SPLINE
SPL {X  -156.487, Y  +349.204, Z    +0.000, E1   +21.338, E3 +359209.083}
SPL {X  -159.136, Y  +365.992, Z    +0.000, E1   +12.463, E3 +359219.841}
SPL {X  -159.799, Y  +374.694, Z    +0.000, E1    +7.504, E3 +359222.945}
SPL {X  -159.976, Y  +380.404, Z    +0.000, E1    +3.959, E3 +359224.478}
SPL {X  -159.990, Y  +384.773, Z    +0.000, E1    +1.003, E3 +359225.373}
SPL {X  -159.990, Y  +387.968, Z    +0.000, E1    -1.448, E3 +359225.941}
SPL {X  -159.990, Y  +391.397, Z    +0.000, E1    -4.422, E3 +359226.565}
SPL {X  -159.990, Y  +395.864, Z    +0.000, E1    -8.712, E3 +359227.653}
SPL {X  -159.990, Y  +401.273, Z    +0.000, E1   -14.176, E3 +359229.381}
SPL {X  -159.990, Y  +411.788, Z    +0.000, E1   -23.693, E3 +359234.924}
SPL {X  -159.990, Y  +438.158, Z    +0.000, E1   -37.630, E3 +359258.201}
SPL {X  -159.990, Y  +468.567, Z    +0.000, E1   -41.922, E3 +359307.545}
SPL {X  -159.990, Y  +474.616, Z    +0.000, E1   -41.909, E3 +359321.874}
SPL {X  -159.990, Y  +478.952, Z    +0.000, E1   -41.885, E3 +359332.172}
SPL {X  -159.990, Y  +484.724, Z    +0.000, E1   -41.943, E3 +359345.724}
SPL {X  -159.990, Y  +492.944, Z    +0.000, E1   -41.952, E3 +359365.143}
SPL {X  -159.990, Y  +499.538, Z    +0.000, E1   -41.904, E3 +359380.802}
SPL {X  -159.990, Y  +504.097, Z    +0.000, E1   -41.897, E3 +359391.590}
SPL {X  -159.990, Y  +509.413, Z    +0.000, E1   -41.921, E3 +359404.126}
SPL {X  -159.990, Y  +516.193, Z    +0.000, E1   -41.932, E3 +359420.142}
SPL {X  -159.990, Y  +521.318, Z    +0.000, E1   -41.891, E3 +359432.316}
SPL {X  -159.990, Y  +526.974, Z    +0.000, E1   -41.950, E3 +359445.605}
SPL {X  -159.990, Y  +533.758, Z    +0.000, E1   -41.910, E3 +359461.708}
SPL {X  -159.990, Y  +539.474, Z    +0.000, E1   -41.912, E3 +359475.235}
SPL {X  -159.990, Y  +544.879, Z    +0.000, E1   -41.899, E3 +359488.046}
SPL {X  -159.990, Y  +550.802, Z    +0.000, E1   -41.920, E3 +359502.028}
SPL {X  -159.990, Y  +556.952, Z    +0.000, E1   -41.911, E3 +359516.567}
SPL {X  -159.990, Y  +562.629, Z    +0.000, E1   -41.910, E3 +359529.985}
SPL {X  -159.990, Y  +567.682, Z    +0.000, E1   -41.901, E3 +359541.944}
SPL {X  -159.990, Y  +572.912, Z    +0.000, E1   -41.914, E3 +359554.291}
SPL {X  -159.990, Y  +578.863, Z    +0.000, E1   -41.918, E3 +359568.355}
SPL {X  -159.990, Y  +584.320, Z    +0.000, E1   -41.901, E3 +359581.302}
SPL {X  -159.990, Y  +589.217, Z    +0.000, E1   -41.901, E3 +359592.875}
SPL {X  -159.990, Y  +594.252, Z    +0.000, E1   -41.903, E3 +359604.789}
SPL {X  -159.990, Y  +600.237, Z    +0.000, E1   -41.928, E3 +359618.907}
SPL {X  -159.990, Y  +605.518, Z    +0.000, E1   -41.890, E3 +359631.445}
SPL {X  -159.990, Y  +610.545, Z    +0.000, E1   -41.917, E3 +359643.293}
SPL {X  -159.990, Y  +615.720, Z    +0.000, E1   -41.899, E3 +359655.553}
SPL {X  -159.990, Y  +621.417, Z    +0.000, E1   -41.931, E3 +359668.990}
SPL {X  -159.990, Y  +627.900, Z    +0.000, E1   -41.914, E3 +359684.330}
SPL {X  -159.990, Y  +632.270, Z    +0.000, E1   -41.887, E3 +359694.706}
SPL {X  -159.990, Y  +637.009, Z    +0.000, E1   -41.925, E3 +359705.848}
SPL {X  -159.990, Y  +642.624, Z    +0.000, E1   -41.901, E3 +359719.169}
SPL {X  -159.990, Y  +647.782, Z    +0.000, E1   -41.914, E3 +359731.337}
SPL {X  -159.990, Y  +653.094, Z    +0.000, E1   -41.905, E3 +359743.916}
SPL {X  -159.990, Y  +657.893, Z    +0.000, E1   -41.899, E3 +359755.281}
SPL {X  -159.990, Y  +662.516, Z    +0.000, E1   -41.899, E3 +359766.213}
SPL {X  -159.990, Y  +666.974, Z    +0.000, E1   -41.897, E3 +359776.757}
SPL {X  -159.984, Y  +672.859, Z    +0.000, E1   -41.934, E3 +359790.618}
SPL {X  -159.817, Y  +678.937, Z    +0.000, E1   -41.879, E3 +359805.206}
SPL {X  -159.484, Y  +684.213, Z    +0.000, E1   -41.818, E3 +359818.043}
SPL {X  -159.007, Y  +689.209, Z    +0.000, E1   -41.732, E3 +359830.347}
SPL {X  -158.327, Y  +694.511, Z    +0.000, E1   -41.622, E3 +359843.598}
SPL {X  -157.480, Y  +699.729, Z    +0.000, E1   -41.453, E3 +359856.861}
SPL {X  -156.604, Y  +704.242, Z    +0.000, E1   -41.288, E3 +359868.470}
SPL {X  -155.514, Y  +709.078, Z    +0.000, E1   -41.107, E3 +359881.024}
SPL {X  -154.232, Y  +714.035, Z    +0.000, E1   -40.861, E3 +359894.083}
SPL {X  -153.147, Y  +717.790, Z    +0.000, E1   -40.640, E3 +359904.101}
SPL {X  -151.881, Y  +721.788, Z    +0.000, E1   -40.435, E3 +359914.787}
SPL {X  -148.572, Y  +730.857, Z    +0.000, E1   -36.304, E3 +359970.996}
ENDSPLINE

SPLINE
SPL {X  -156.377, Y  +705.307, Z    +0.000, E1   -21.740, E3 +360025.245}
SPL {X  -158.965, Y  +689.585, Z    +0.000, E1   -13.405, E3 +360036.403}
SPL {X  -159.884, Y  +677.314, Z    +0.000, E1    -6.475, E3 +360041.115}
SPL {X  -159.990, Y  +670.142, Z    +0.000, E1    -1.740, E3 +360042.905}
SPL {X  -159.990, Y  +666.629, Z    +0.000, E1    +0.827, E3 +360043.554}
SPL {X  -159.990, Y  +662.407, Z    +0.000, E1    +4.406, E3 +360044.405}
SPL {X  -159.990, Y  +655.884, Z    +0.000, E1   +10.601, E3 +360046.270}
SPL {X  -159.990, Y  +643.833, Z    +0.000, E1   +21.883, E3 +360051.899}
SPL {X  -159.990, Y  +617.235, Z    +0.000, E1   +36.481, E3 +360075.799}
SPL {X  -159.990, Y  +586.905, Z    +0.000, E1   +41.264, E3 +360124.776}
SPL {X  -159.990, Y  +581.111, Z    +0.000, E1   +41.245, E3 +360138.829}
SPL {X  -159.990, Y  +576.269, Z    +0.000, E1   +41.239, E3 +360150.557}
SPL {X  -159.990, Y  +571.714, Z    +0.000, E1   +41.240, E3 +360161.585}
SPL {X  -159.990, Y  +567.050, Z    +0.000, E1   +41.238, E3 +360172.872}
SPL {X  -159.990, Y  +561.959, Z    +0.000, E1   +41.251, E3 +360185.170}
SPL {X  -159.990, Y  +557.719, Z    +0.000, E1   +41.226, E3 +360195.473}
SPL {X  -159.990, Y  +554.148, Z    +0.000, E1   +41.237, E3 +360204.088}
SPL {X  -159.990, Y  +548.812, Z    +0.000, E1   +41.263, E3 +360216.963}
SPL {X  -159.990, Y  +543.804, Z    +0.000, E1   +41.237, E3 +360229.127}
SPL {X  -159.990, Y  +538.952, Z    +0.000, E1   +41.247, E3 +360240.875}
SPL {X  -159.990, Y  +534.225, Z    +0.000, E1   +41.236, E3 +360252.308}
SPL {X  -159.990, Y  +529.136, Z    +0.000, E1   +41.262, E3 +360264.584}
SPL {X  -159.990, Y  +522.690, Z    +0.000, E1   +41.265, E3 +360280.183}
SPL {X  -159.990, Y  +516.698, Z    +0.000, E1   +41.259, E3 +360294.658}
SPL {X  -159.990, Y  +510.896, Z    +0.000, E1   +41.267, E3 +360308.675}
SPL {X  -159.990, Y  +505.215, Z    +0.000, E1   +41.261, E3 +360322.435}
SPL {X  -159.990, Y  +500.102, Z    +0.000, E1   +41.251, E3 +360334.819}
SPL {X  -159.990, Y  +495.023, Z    +0.000, E1   +41.263, E3 +360347.067}
SPL {X  -159.990, Y  +479.011, Z    +0.000, E1   +45.740, E3 +360356.449}
SPL {X  -159.990, Y  +471.379, Z    +0.000, E1   +46.435, E3 +360368.065}
SPL {X  -159.990, Y  +466.895, Z    +0.000, E1   +45.533, E3 +360382.470}
SPL {X  -159.990, Y  +462.409, Z    +0.000, E1   +44.664, E3 +360397.245}
SPL {X  -159.990, Y  +458.229, Z    +0.000, E1   +43.579, E3 +360412.727}
SPL {X  -159.990, Y  +453.434, Z    +0.000, E1   +43.227, E3 +360425.501}
SPL {X  -159.990, Y  +448.702, Z    +0.000, E1   +43.218, E3 +360436.223}
SPL {X  -159.990, Y  +444.476, Z    +0.000, E1   +43.219, E3 +360445.761}
SPL {X  -159.990, Y  +440.246, Z    +0.000, E1   +43.217, E3 +360455.319}
SPL {X  -159.990, Y  +434.411, Z    +0.000, E1   +43.246, E3 +360468.449}
SPL {X  -159.990, Y  +429.216, Z    +0.000, E1   +43.210, E3 +360480.222}
SPL {X  -159.990, Y  +424.433, Z    +0.000, E1   +43.237, E3 +360490.970}
SPL {X  -159.990, Y  +419.466, Z    +0.000, E1   +43.217, E3 +360502.209}
SPL {X  -159.990, Y  +414.585, Z    +0.000, E1   +43.233, E3 +360513.201}
SPL {X  -159.990, Y  +409.927, Z    +0.000, E1   +43.217, E3 +360523.733}
SPL {X  -159.990, Y  +405.428, Z    +0.000, E1   +43.230, E3 +360533.891}
SPL {X  -159.990, Y  +398.518, Z    +0.000, E1   +43.261, E3 +360549.445}
SPL {X  -159.990, Y  +392.163, Z    +0.000, E1   +43.223, E3 +360563.845}
SPL {X  -159.990, Y  +387.342, Z    +0.000, E1   +43.224, E3 +360574.723}
SPL {X  -159.990, Y  +382.548, Z    +0.000, E1   +43.224, E3 +360585.546}
SPL {X  -159.922, Y  +377.835, Z    +0.000, E1   +43.211, E3 +360596.262}
SPL {X  -159.712, Y  +373.072, Z    +0.000, E1   +43.177, E3 +360607.228}
SPL {X  -159.289, Y  +367.537, Z    +0.000, E1   +43.118, E3 +360620.140}
SPL {X  -158.730, Y  +362.464, Z    +0.000, E1   +43.003, E3 +360632.172}
SPL {X  -158.182, Y  +358.518, Z    +0.000, E1   +42.902, E3 +360641.650}
SPL {X  -157.507, Y  +354.423, Z    +0.000, E1   +42.786, E3 +360651.596}
SPL {X  -156.676, Y  +350.104, Z    +0.000, E1   +42.637, E3 +360662.201}
SPL {X  -155.807, Y  +346.154, Z    +0.000, E1   +42.470, E3 +360672.028}
SPL {X  -154.777, Y  +341.993, Z    +0.000, E1   +42.302, E3 +360682.453}
SPL {X  -153.585, Y  +337.686, Z    +0.000, E1   +42.062, E3 +360693.429}
SPL {X  -152.412, Y  +333.846, Z    +0.000, E1   +41.856, E3 +360703.271}
SPL {X  -151.009, Y  +329.651, Z    +0.000, E1   +41.581, E3 +360714.171}
SPL {X  -148.356, Y  +322.607, Z    +0.000, E1   +36.121, E3 +360774.647}
ENDSPLINE

SPLINE
SPL {X  -156.487, Y  +349.204, Z    +0.000, E1   +21.338, E3 +360829.773}
SPL {X  -159.136, Y  +365.992, Z    +0.000, E1   +12.463, E3 +360840.531}
SPL {X  -159.799, Y  +374.694, Z    +0.000, E1    +7.504, E3 +360843.635}
SPL {X  -159.976, Y  +380.404, Z    +0.000, E1    +3.959, E3 +360845.168}
SPL {X  -159.990, Y  +384.773, Z    +0.000, E1    +1.003, E3 +360846.062}
SPL {X  -159.990, Y  +387.968, Z    +0.000, E1    -1.448, E3 +360846.631}
SPL {X  -159.990, Y  +391.397, Z    +0.000, E1    -4.422, E3 +360847.255}
SPL {X  -159.990, Y  +395.864, Z    +0.000, E1    -8.712, E3 +360848.343}
SPL {X  -159.990, Y  +401.273, Z    +0.000, E1   -14.176, E3 +360850.070}
SPL {X  -159.990, Y  +409.369, Z    +0.000, E1   -21.807, E3 +360853.862}
SPL {X  -159.990, Y  +436.107, Z    +0.000, E1   -36.921, E3 +360876.787}
SPL {X  -159.990, Y  +465.724, Z    +0.000, E1   -41.883, E3 +360921.586}
SPL {X  -159.990, Y  +470.837, Z    +0.000, E1   -41.927, E3 +360933.600}
SPL {X  -159.990, Y  +477.498, Z    +0.000, E1   -41.916, E3 +360949.375}
SPL {X  -159.990, Y  +483.140, Z    +0.000, E1   -41.902, E3 +360962.731}
SPL {X  -159.990, Y  +488.618, Z    +0.000, E1   -41.913, E3 +360975.663}
SPL {X  -159.990, Y  +494.299, Z    +0.000, E1   -41.910, E3 +360989.097}
SPL {X  -159.990, Y  +499.538, Z    +0.000, E1   -41.904, E3 +361001.491}
SPL {X  -159.990, Y  +505.259, Z    +0.000, E1   -41.922, E3 +361014.991}
SPL {X  -159.990, Y  +511.862, Z    +0.000, E1   -41.927, E3 +361030.601}
SPL {X  -159.990, Y  +519.146, Z    +0.000, E1   -41.942, E3 +361047.795}
SPL {X  -159.990, Y  +526.974, Z    +0.000, E1   -41.950, E3 +361066.295}
SPL {X  -159.990, Y  +533.758, Z    +0.000, E1   -41.910, E3 +361082.397}
SPL {X  -159.990, Y  +539.474, Z    +0.000, E1   -41.912, E3 +361095.925}
SPL {X  -159.990, Y  +544.879, Z    +0.000, E1   -41.899, E3 +361108.736}
SPL {X  -159.990, Y  +550.802, Z    +0.000, E1   -41.920, E3 +361122.717}
SPL {X  -159.990, Y  +556.952, Z    +0.000, E1   -41.911, E3 +361137.257}
SPL {X  -159.990, Y  +562.629, Z    +0.000, E1   -41.910, E3 +361150.675}
SPL {X  -159.990, Y  +567.682, Z    +0.000, E1   -41.901, E3 +361162.634}
SPL {X  -159.990, Y  +572.912, Z    +0.000, E1   -41.914, E3 +361174.981}
SPL {X  -159.990, Y  +578.863, Z    +0.000, E1   -41.918, E3 +361189.045}
SPL {X  -159.990, Y  +584.320, Z    +0.000, E1   -41.901, E3 +361201.992}
SPL {X  -159.990, Y  +589.217, Z    +0.000, E1   -41.901, E3 +361213.564}
SPL {X  -159.990, Y  +594.252, Z    +0.000, E1   -41.903, E3 +361225.479}
SPL {X  -159.990, Y  +598.793, Z    +0.000, E1   -41.896, E3 +361236.233}
SPL {X  -159.990, Y  +604.215, Z    +0.000, E1   -41.919, E3 +361249.013}
SPL {X  -159.990, Y  +609.216, Z    +0.000, E1   -41.890, E3 +361260.881}
SPL {X  -159.990, Y  +614.570, Z    +0.000, E1   -41.926, E3 +361273.486}
SPL {X  -159.990, Y  +620.005, Z    +0.000, E1   -41.900, E3 +361286.376}
SPL {X  -159.990, Y  +624.919, Z    +0.000, E1   -41.912, E3 +361297.983}
SPL {X  -159.990, Y  +630.816, Z    +0.000, E1   -41.915, E3 +361311.912}
SPL {X  -159.990, Y  +637.009, Z    +0.000, E1   -41.925, E3 +361326.538}
SPL {X  -159.990, Y  +642.624, Z    +0.000, E1   -41.901, E3 +361339.858}
SPL {X  -159.990, Y  +647.782, Z    +0.000, E1   -41.914, E3 +361352.027}
SPL {X  -159.990, Y  +653.094, Z    +0.000, E1   -41.905, E3 +361364.605}
SPL {X  -159.990, Y  +657.893, Z    +0.000, E1   -41.899, E3 +361375.971}
SPL {X  -159.990, Y  +662.516, Z    +0.000, E1   -41.899, E3 +361386.902}
SPL {X  -159.990, Y  +666.974, Z    +0.000, E1   -41.897, E3 +361397.447}
SPL {X  -159.984, Y  +672.859, Z    +0.000, E1   -41.934, E3 +361411.308}
SPL {X  -159.817, Y  +678.937, Z    +0.000, E1   -41.879, E3 +361425.896}
SPL {X  -159.484, Y  +684.213, Z    +0.000, E1   -41.818, E3 +361438.732}
SPL {X  -159.007, Y  +689.209, Z    +0.000, E1   -41.732, E3 +361451.037}
SPL {X  -158.327, Y  +694.511, Z    +0.000, E1   -41.622, E3 +361464.288}
SPL {X  -157.480, Y  +699.729, Z    +0.000, E1   -41.453, E3 +361477.551}
SPL {X  -156.604, Y  +704.242, Z    +0.000, E1   -41.288, E3 +361489.160}
SPL {X  -155.514, Y  +709.078, Z    +0.000, E1   -41.107, E3 +361501.713}
SPL {X  -154.232, Y  +714.035, Z    +0.000, E1   -40.861, E3 +361514.772}
SPL {X  -153.147, Y  +717.790, Z    +0.000, E1   -40.640, E3 +361524.791}
SPL {X  -151.881, Y  +721.788, Z    +0.000, E1   -40.435, E3 +361535.477}
SPL {X  -148.572, Y  +730.857, Z    +0.000, E1   -36.304, E3 +361591.686}
ENDSPLINE

SPLINE
SPL {X  -156.377, Y  +705.307, Z    +0.000, E1   -21.740, E3 +361645.935}
SPL {X  -158.965, Y  +689.585, Z    +0.000, E1   -13.405, E3 +361657.092}
SPL {X  -159.884, Y  +677.314, Z    +0.000, E1    -6.475, E3 +361661.805}
SPL {X  -159.990, Y  +670.142, Z    +0.000, E1    -1.740, E3 +361663.594}
SPL {X  -159.990, Y  +666.629, Z    +0.000, E1    +0.827, E3 +361664.244}
SPL {X  -159.990, Y  +662.407, Z    +0.000, E1    +4.406, E3 +361665.094}
SPL {X  -159.990, Y  +655.884, Z    +0.000, E1   +10.601, E3 +361666.960}
SPL {X  -159.990, Y  +643.833, Z    +0.000, E1   +21.883, E3 +361672.589}
SPL {X  -159.990, Y  +617.235, Z    +0.000, E1   +36.481, E3 +361696.489}
SPL {X  -159.990, Y  +586.905, Z    +0.000, E1   +41.264, E3 +361745.465}
SPL {X  -159.990, Y  +581.111, Z    +0.000, E1   +41.245, E3 +361759.519}
SPL {X  -159.990, Y  +576.269, Z    +0.000, E1   +41.239, E3 +361771.247}
SPL {X  -159.990, Y  +571.714, Z    +0.000, E1   +41.240, E3 +361782.275}
SPL {X  -159.990, Y  +567.050, Z    +0.000, E1   +41.238, E3 +361793.561}
SPL {X  -159.990, Y  +561.959, Z    +0.000, E1   +41.251, E3 +361805.860}
SPL {X  -159.990, Y  +555.553, Z    +0.000, E1   +41.273, E3 +361821.328}
SPL {X  -159.990, Y  +549.897, Z    +0.000, E1   +41.240, E3 +361835.058}
SPL {X  -159.990, Y  +544.775, Z    +0.000, E1   +41.260, E3 +361847.433}
SPL {X  -159.990, Y  +538.952, Z    +0.000, E1   +41.247, E3 +361861.564}
SPL {X  -159.990, Y  +534.225, Z    +0.000, E1   +41.236, E3 +361872.997}
SPL {X  -159.990, Y  +529.136, Z    +0.000, E1   +41.262, E3 +361885.273}
SPL {X  -159.990, Y  +524.776, Z    +0.000, E1   +41.225, E3 +361895.887}
SPL {X  -159.990, Y  +521.454, Z    +0.000, E1   +41.236, E3 +361903.909}
SPL {X  -159.990, Y  +515.605, Z    +0.000, E1   +41.288, E3 +361917.948}
SPL {X  -159.990, Y  +509.898, Z    +0.000, E1   +41.246, E3 +361931.809}
SPL {X  -159.990, Y  +505.215, Z    +0.000, E1   +41.261, E3 +361943.125}
SPL {X  -159.990, Y  +500.102, Z    +0.000, E1   +41.251, E3 +361955.508}
SPL {X  -159.990, Y  +495.023, Z    +0.000, E1   +41.263, E3 +361967.757}
SPL {X  -159.990, Y  +479.011, Z    +0.000, E1   +45.740, E3 +361977.139}
SPL {X  -159.990, Y  +471.379, Z    +0.000, E1   +46.435, E3 +361988.754}
SPL {X  -159.990, Y  +465.881, Z    +0.000, E1   +45.385, E3 +362006.357}
SPL {X  -159.990, Y  +461.571, Z    +0.000, E1   +44.440, E3 +362020.883}
SPL {X  -159.990, Y  +458.229, Z    +0.000, E1   +43.579, E3 +362033.416}
SPL {X  -159.990, Y  +453.434, Z    +0.000, E1   +43.227, E3 +362046.191}
SPL {X  -159.990, Y  +448.702, Z    +0.000, E1   +43.218, E3 +362056.913}
SPL {X  -159.990, Y  +442.224, Z    +0.000, E1   +43.270, E3 +362071.463}
SPL {X  -159.990, Y  +435.724, Z    +0.000, E1   +43.218, E3 +362086.221}
SPL {X  -159.990, Y  +430.527, Z    +0.000, E1   +43.236, E3 +362097.910}
SPL {X  -159.990, Y  +424.433, Z    +0.000, E1   +43.237, E3 +362111.659}
SPL {X  -159.990, Y  +419.466, Z    +0.000, E1   +43.217, E3 +362122.899}
SPL {X  -159.990, Y  +414.585, Z    +0.000, E1   +43.233, E3 +362133.891}
SPL {X  -159.990, Y  +409.927, Z    +0.000, E1   +43.217, E3 +362144.422}
SPL {X  -159.990, Y  +405.428, Z    +0.000, E1   +43.230, E3 +362154.581}
SPL {X  -159.990, Y  +401.033, Z    +0.000, E1   +43.209, E3 +362164.535}
SPL {X  -159.990, Y  +396.968, Z    +0.000, E1   +43.221, E3 +362173.693}
SPL {X  -159.990, Y  +392.163, Z    +0.000, E1   +43.223, E3 +362184.535}
SPL {X  -159.990, Y  +387.342, Z    +0.000, E1   +43.224, E3 +362195.412}
SPL {X  -159.990, Y  +382.548, Z    +0.000, E1   +43.224, E3 +362206.235}
SPL {X  -159.922, Y  +377.835, Z    +0.000, E1   +43.211, E3 +362216.952}
SPL {X  -159.712, Y  +373.072, Z    +0.000, E1   +43.177, E3 +362227.918}
SPL {X  -159.289, Y  +367.537, Z    +0.000, E1   +43.118, E3 +362240.830}
SPL {X  -158.730, Y  +362.464, Z    +0.000, E1   +43.003, E3 +362252.862}
SPL {X  -158.182, Y  +358.518, Z    +0.000, E1   +42.902, E3 +362262.340}
SPL {X  -157.507, Y  +354.423, Z    +0.000, E1   +42.786, E3 +362272.285}
SPL {X  -156.676, Y  +350.104, Z    +0.000, E1   +42.637, E3 +362282.891}
SPL {X  -155.807, Y  +346.154, Z    +0.000, E1   +42.470, E3 +362292.718}
SPL {X  -154.777, Y  +341.993, Z    +0.000, E1   +42.302, E3 +362303.143}
SPL {X  -153.585, Y  +337.686, Z    +0.000, E1   +42.062, E3 +362314.118}
SPL {X  -152.412, Y  +333.846, Z    +0.000, E1   +41.856, E3 +362323.961}
SPL {X  -151.009, Y  +329.651, Z    +0.000, E1   +41.581, E3 +362334.861}
SPL {X  -148.356, Y  +322.607, Z    +0.000, E1   +36.121, E3 +362395.336}
ENDSPLINE

SPLINE
SPL {X  -156.487, Y  +349.204, Z    +0.000, E1   +21.338, E3 +362450.462}
SPL {X  -159.136, Y  +365.992, Z    +0.000, E1   +12.463, E3 +362461.221}
SPL {X  -159.799, Y  +374.694, Z    +0.000, E1    +7.504, E3 +362464.324}
SPL {X  -159.976, Y  +380.404, Z    +0.000, E1    +3.959, E3 +362465.857}
SPL {X  -159.990, Y  +384.773, Z    +0.000, E1    +1.003, E3 +362466.752}
SPL {X  -159.990, Y  +387.968, Z    +0.000, E1    -1.448, E3 +362467.320}
SPL {X  -159.990, Y  +391.397, Z    +0.000, E1    -4.422, E3 +362467.944}
SPL {X  -159.990, Y  +395.864, Z    +0.000, E1    -8.712, E3 +362469.033}
SPL {X  -159.990, Y  +401.273, Z    +0.000, E1   -14.176, E3 +362470.760}
SPL {X  -159.990, Y  +409.369, Z    +0.000, E1   -21.807, E3 +362474.552}
SPL {X  -159.990, Y  +436.107, Z    +0.000, E1   -36.921, E3 +362497.477}
SPL {X  -159.990, Y  +468.567, Z    +0.000, E1   -41.922, E3 +362548.924}
SPL {X  -159.990, Y  +474.616, Z    +0.000, E1   -41.909, E3 +362563.254}
SPL {X  -159.990, Y  +481.610, Z    +0.000, E1   -41.947, E3 +362579.740}
SPL {X  -159.990, Y  +488.618, Z    +0.000, E1   -41.913, E3 +362596.353}
SPL {X  -159.990, Y  +494.299, Z    +0.000, E1   -41.910, E3 +362609.787}
SPL {X  -159.990, Y  +499.538, Z    +0.000, E1   -41.904, E3 +362622.181}
SPL {X  -159.990, Y  +505.259, Z    +0.000, E1   -41.922, E3 +362635.680}
SPL {X  -159.990, Y  +511.862, Z    +0.000, E1   -41.927, E3 +362651.291}
SPL {X  -159.990, Y  +519.146, Z    +0.000, E1   -41.942, E3 +362668.484}
SPL {X  -159.990, Y  +526.974, Z    +0.000, E1   -41.950, E3 +362686.984}
SPL {X  -159.990, Y  +533.758, Z    +0.000, E1   -41.910, E3 +362703.087}
SPL {X  -159.990, Y  +539.474, Z    +0.000, E1   -41.912, E3 +362716.614}
SPL {X  -159.990, Y  +546.447, Z    +0.000, E1   -41.939, E3 +362733.077}
SPL {X  -159.990, Y  +552.220, Z    +0.000, E1   -41.887, E3 +362746.811}
SPL {X  -159.990, Y  +556.952, Z    +0.000, E1   -41.911, E3 +362757.946}
SPL {X  -159.990, Y  +562.629, Z    +0.000, E1   -41.910, E3 +362771.364}
SPL {X  -159.990, Y  +567.682, Z    +0.000, E1   -41.901, E3 +362783.323}
SPL {X  -159.990, Y  +574.350, Z    +0.000, E1   -41.955, E3 +362799.009}
SPL {X  -159.990, Y  +580.118, Z    +0.000, E1   -41.891, E3 +362812.745}
SPL {X  -159.990, Y  +584.320, Z    +0.000, E1   -41.901, E3 +362822.681}
SPL {X  -159.990, Y  +589.217, Z    +0.000, E1   -41.901, E3 +362834.254}
SPL {X  -159.990, Y  +594.252, Z    +0.000, E1   -41.903, E3 +362846.169}
SPL {X  -159.990, Y  +600.237, Z    +0.000, E1   -41.928, E3 +362860.286}
SPL {X  -159.990, Y  +605.518, Z    +0.000, E1   -41.890, E3 +362872.824}
SPL {X  -159.990, Y  +610.545, Z    +0.000, E1   -41.917, E3 +362884.673}
SPL {X  -159.990, Y  +615.720, Z    +0.000, E1   -41.899, E3 +362896.933}
SPL {X  -159.990, Y  +620.005, Z    +0.000, E1   -41.900, E3 +362907.066}
SPL {X  -159.990, Y  +624.919, Z    +0.000, E1   -41.912, E3 +362918.673}
SPL {X  -159.990, Y  +629.282, Z    +0.000, E1   -41.888, E3 +362929.013}
SPL {X  -159.990, Y  +634.411, Z    +0.000, E1   -41.931, E3 +362941.078}
SPL {X  -159.990, Y  +641.479, Z    +0.000, E1   -41.931, E3 +362957.795}
SPL {X  -159.990, Y  +647.782, Z    +0.000, E1   -41.914, E3 +362972.717}
SPL {X  -159.990, Y  +653.094, Z    +0.000, E1   -41.905, E3 +362985.295}
SPL {X  -159.990, Y  +657.893, Z    +0.000, E1   -41.899, E3 +362996.660}
SPL {X  -159.990, Y  +662.516, Z    +0.000, E1   -41.899, E3 +363007.592}
SPL {X  -159.990, Y  +668.411, Z    +0.000, E1   -41.929, E3 +363021.486}
SPL {X  -159.968, Y  +674.139, Z    +0.000, E1   -41.898, E3 +363035.089}
SPL {X  -159.817, Y  +678.937, Z    +0.000, E1   -41.879, E3 +363046.586}
SPL {X  -159.484, Y  +684.213, Z    +0.000, E1   -41.818, E3 +363059.422}
SPL {X  -159.007, Y  +689.209, Z    +0.000, E1   -41.732, E3 +363071.727}
SPL {X  -158.327, Y  +694.511, Z    +0.000, E1   -41.622, E3 +363084.978}
SPL {X  -157.480, Y  +699.729, Z    +0.000, E1   -41.453, E3 +363098.241}
SPL {X  -156.604, Y  +704.242, Z    +0.000, E1   -41.288, E3 +363109.849}
SPL {X  -155.831, Y  +707.744, Z    +0.000, E1   -41.132, E3 +363118.969}
SPL {X  -155.167, Y  +710.488, Z    +0.000, E1   -41.008, E3 +363126.147}
SPL {X  -154.232, Y  +714.035, Z    +0.000, E1   -40.861, E3 +363135.462}
SPL {X  -153.147, Y  +717.790, Z    +0.000, E1   -40.640, E3 +363145.480}
SPL {X  -151.881, Y  +721.788, Z    +0.000, E1   -40.435, E3 +363156.167}
SPL {X  -148.572, Y  +730.857, Z    +0.000, E1   -36.304, E3 +363212.376}
ENDSPLINE

SPLINE
SPL {X  -156.377, Y  +705.307, Z    +0.000, E1   -21.740, E3 +363266.624}
SPL {X  -159.301, Y  +686.331, Z    +0.000, E1   -11.648, E3 +363279.269}
SPL {X  -159.936, Y  +675.651, Z    +0.000, E1    -5.377, E3 +363282.985}
SPL {X  -159.990, Y  +670.142, Z    +0.000, E1    -1.740, E3 +363284.284}
SPL {X  -159.990, Y  +666.629, Z    +0.000, E1    +0.827, E3 +363284.933}
SPL {X  -159.990, Y  +662.407, Z    +0.000, E1    +4.406, E3 +363285.784}
SPL {X  -159.990, Y  +655.884, Z    +0.000, E1   +10.601, E3 +363287.649}
SPL {X  -159.990, Y  +643.833, Z    +0.000, E1   +21.883, E3 +363293.278}
SPL {X  -159.990, Y  +617.235, Z    +0.000, E1   +36.481, E3 +363317.178}
SPL {X  -159.990, Y  +586.905, Z    +0.000, E1   +41.264, E3 +363366.155}
SPL {X  -159.990, Y  +581.111, Z    +0.000, E1   +41.245, E3 +363380.209}
SPL {X  -159.990, Y  +576.269, Z    +0.000, E1   +41.239, E3 +363391.936}
SPL {X  -159.990, Y  +571.714, Z    +0.000, E1   +41.240, E3 +363402.964}
SPL {X  -159.990, Y  +567.050, Z    +0.000, E1   +41.238, E3 +363414.251}
SPL {X  -159.990, Y  +561.959, Z    +0.000, E1   +41.251, E3 +363426.550}
SPL {X  -159.990, Y  +555.553, Z    +0.000, E1   +41.273, E3 +363442.018}
SPL {X  -159.990, Y  +549.897, Z    +0.000, E1   +41.240, E3 +363455.748}
SPL {X  -159.990, Y  +544.775, Z    +0.000, E1   +41.260, E3 +363468.123}
SPL {X  -159.990, Y  +538.952, Z    +0.000, E1   +41.247, E3 +363482.254}
SPL {X  -159.990, Y  +534.225, Z    +0.000, E1   +41.236, E3 +363493.687}
SPL {X  -159.990, Y  +529.136, Z    +0.000, E1   +41.262, E3 +363505.963}
SPL {X  -159.990, Y  +522.690, Z    +0.000, E1   +41.265, E3 +363521.563}
SPL {X  -159.990, Y  +516.698, Z    +0.000, E1   +41.259, E3 +363536.037}
SPL {X  -159.990, Y  +510.896, Z    +0.000, E1   +41.267, E3 +363550.055}
SPL {X  -159.990, Y  +505.215, Z    +0.000, E1   +41.261, E3 +363563.815}
SPL {X  -159.990, Y  +500.102, Z    +0.000, E1   +41.251, E3 +363576.198}
SPL {X  -159.990, Y  +495.023, Z    +0.000, E1   +41.263, E3 +363588.447}
SPL {X  -159.990, Y  +479.011, Z    +0.000, E1   +45.740, E3 +363597.829}
SPL {X  -159.990, Y  +471.379, Z    +0.000, E1   +46.435, E3 +363609.444}
SPL {X  -159.990, Y  +465.881, Z    +0.000, E1   +45.385, E3 +363627.047}
SPL {X  -159.990, Y  +461.571, Z    +0.000, E1   +44.440, E3 +363641.572}
SPL {X  -159.990, Y  +458.229, Z    +0.000, E1   +43.579, E3 +363654.106}
SPL {X  -159.990, Y  +453.434, Z    +0.000, E1   +43.227, E3 +363666.880}
SPL {X  -159.990, Y  +448.702, Z    +0.000, E1   +43.218, E3 +363677.602}
SPL {X  -159.990, Y  +444.476, Z    +0.000, E1   +43.219, E3 +363687.141}
SPL {X  -159.990, Y  +440.246, Z    +0.000, E1   +43.217, E3 +363696.698}
SPL {X  -159.990, Y  +434.411, Z    +0.000, E1   +43.246, E3 +363709.828}
SPL {X  -159.990, Y  +429.216, Z    +0.000, E1   +43.210, E3 +363721.601}
SPL {X  -159.990, Y  +424.433, Z    +0.000, E1   +43.237, E3 +363732.349}
SPL {X  -159.990, Y  +419.466, Z    +0.000, E1   +43.217, E3 +363743.588}
SPL {X  -159.990, Y  +414.585, Z    +0.000, E1   +43.233, E3 +363754.580}
SPL {X  -159.990, Y  +409.927, Z    +0.000, E1   +43.217, E3 +363765.112}
SPL {X  -159.990, Y  +405.428, Z    +0.000, E1   +43.230, E3 +363775.270}
SPL {X  -159.990, Y  +398.518, Z    +0.000, E1   +43.261, E3 +363790.825}
SPL {X  -159.990, Y  +392.163, Z    +0.000, E1   +43.223, E3 +363805.225}
SPL {X  -159.990, Y  +387.342, Z    +0.000, E1   +43.224, E3 +363816.102}
SPL {X  -159.990, Y  +382.548, Z    +0.000, E1   +43.224, E3 +363826.925}
SPL {X  -159.922, Y  +377.835, Z    +0.000, E1   +43.211, E3 +363837.642}
SPL {X  -159.712, Y  +373.072, Z    +0.000, E1   +43.177, E3 +363848.608}
SPL {X  -159.289, Y  +367.537, Z    +0.000, E1   +43.118, E3 +363861.519}
SPL {X  -158.730, Y  +362.464, Z    +0.000, E1   +43.003, E3 +363873.551}
SPL {X  -158.182, Y  +358.518, Z    +0.000, E1   +42.902, E3 +363883.030}
SPL {X  -157.507, Y  +354.423, Z    +0.000, E1   +42.786, E3 +363892.975}
SPL {X  -156.676, Y  +350.104, Z    +0.000, E1   +42.637, E3 +363903.580}
SPL {X  -155.807, Y  +346.154, Z    +0.000, E1   +42.470, E3 +363913.407}
SPL {X  -154.777, Y  +341.993, Z    +0.000, E1   +42.302, E3 +363923.833}
SPL {X  -153.585, Y  +337.686, Z    +0.000, E1   +42.062, E3 +363934.808}
SPL {X  -152.412, Y  +333.846, Z    +0.000, E1   +41.856, E3 +363944.651}
SPL {X  -151.009, Y  +329.651, Z    +0.000, E1   +41.581, E3 +363955.550}
SPL {X  -148.356, Y  +322.607, Z    +0.000, E1   +36.121, E3 +364016.026}
ENDSPLINE

SPLINE
SPL {X  -156.487, Y  +349.204, Z    +0.000, E1   +21.338, E3 +364071.152}
SPL {X  -159.136, Y  +365.992, Z    +0.000, E1   +12.463, E3 +364081.910}
SPL {X  -159.799, Y  +374.694, Z    +0.000, E1    +7.504, E3 +364085.014}
SPL {X  -159.976, Y  +380.404, Z    +0.000, E1    +3.959, E3 +364086.547}
SPL {X  -159.990, Y  +384.773, Z    +0.000, E1    +1.003, E3 +364087.442}
SPL {X  -159.990, Y  +387.968, Z    +0.000, E1    -1.448, E3 +364088.010}
SPL {X  -159.990, Y  +391.397, Z    +0.000, E1    -4.422, E3 +364088.634}
SPL {X  -159.990, Y  +395.864, Z    +0.000, E1    -8.712, E3 +364089.722}
SPL {X  -159.990, Y  +401.273, Z    +0.000, E1   -14.176, E3 +364091.450}
SPL {X  -159.990, Y  +409.369, Z    +0.000, E1   -21.807, E3 +364095.242}
SPL {X  -159.990, Y  +436.107, Z    +0.000, E1   -36.921, E3 +364118.167}
SPL {X  -159.990, Y  +469.969, Z    +0.000, E1   -41.961, E3 +364172.871}
SPL {X  -159.990, Y  +477.498, Z    +0.000, E1   -41.916, E3 +364190.755}
SPL {X  -159.990, Y  +483.140, Z    +0.000, E1   -41.902, E3 +364204.111}
SPL {X  -159.990, Y  +488.618, Z    +0.000, E1   -41.913, E3 +364217.042}
SPL {X  -159.990, Y  +494.299, Z    +0.000, E1   -41.910, E3 +364230.476}
SPL {X  -159.990, Y  +499.538, Z    +0.000, E1   -41.904, E3 +364242.871}
SPL {X  -159.990, Y  +504.097, Z    +0.000, E1   -41.897, E3 +364253.659}
SPL {X  -159.990, Y  +509.413, Z    +0.000, E1   -41.921, E3 +364266.195}
SPL {X  -159.990, Y  +513.834, Z    +0.000, E1   -41.885, E3 +364276.708}
SPL {X  -159.990, Y  +517.450, Z    +0.000, E1   -41.901, E3 +364285.228}
SPL {X  -159.990, Y  +523.027, Z    +0.000, E1   -41.926, E3 +364298.372}
SPL {X  -159.990, Y  +528.611, Z    +0.000, E1   -41.900, E3 +364311.627}
SPL {X  -159.990, Y  +533.758, Z    +0.000, E1   -41.910, E3 +364323.776}
SPL {X  -159.990, Y  +539.474, Z    +0.000, E1   -41.912, E3 +364337.304}
SPL {X  -159.990, Y  +544.879, Z    +0.000, E1   -41.899, E3 +364350.115}
SPL {X  -159.990, Y  +550.802, Z    +0.000, E1   -41.920, E3 +364364.097}
SPL {X  -159.990, Y  +556.952, Z    +0.000, E1   -41.911, E3 +364378.636}
SPL {X  -159.990, Y  +562.629, Z    +0.000, E1   -41.910, E3 +364392.054}
SPL {X  -159.990, Y  +567.682, Z    +0.000, E1   -41.901, E3 +364404.013}
SPL {X  -159.990, Y  +572.912, Z    +0.000, E1   -41.914, E3 +364416.360}
SPL {X  -159.990, Y  +578.863, Z    +0.000, E1   -41.918, E3 +364430.424}
SPL {X  -159.990, Y  +584.320, Z    +0.000, E1   -41.901, E3 +364443.371}
SPL {X  -159.990, Y  +589.217, Z    +0.000, E1   -41.901, E3 +364454.944}
SPL {X  -159.990, Y  +594.252, Z    +0.000, E1   -41.903, E3 +364466.858}
SPL {X  -159.990, Y  +598.793, Z    +0.000, E1   -41.896, E3 +364477.612}
SPL {X  -159.990, Y  +604.215, Z    +0.000, E1   -41.919, E3 +364490.392}
SPL {X  -159.990, Y  +610.545, Z    +0.000, E1   -41.917, E3 +364505.362}
SPL {X  -159.990, Y  +615.720, Z    +0.000, E1   -41.899, E3 +364517.622}
SPL {X  -159.990, Y  +620.005, Z    +0.000, E1   -41.900, E3 +364527.755}
SPL {X  -159.990, Y  +624.919, Z    +0.000, E1   -41.912, E3 +364539.363}
SPL {X  -159.990, Y  +630.816, Z    +0.000, E1   -41.915, E3 +364553.292}
SPL {X  -159.990, Y  +637.009, Z    +0.000, E1   -41.925, E3 +364567.917}
SPL {X  -159.990, Y  +642.624, Z    +0.000, E1   -41.901, E3 +364581.238}
SPL {X  -159.990, Y  +647.782, Z    +0.000, E1   -41.914, E3 +364593.406}
SPL {X  -159.990, Y  +653.094, Z    +0.000, E1   -41.905, E3 +364605.985}
SPL {X  -159.990, Y  +657.893, Z    +0.000, E1   -41.899, E3 +364617.350}
SPL {X  -159.990, Y  +662.516, Z    +0.000, E1   -41.899, E3 +364628.282}
SPL {X  -159.990, Y  +668.411, Z    +0.000, E1   -41.929, E3 +364642.175}
SPL {X  -159.968, Y  +674.139, Z    +0.000, E1   -41.898, E3 +364655.779}
SPL {X  -159.817, Y  +678.937, Z    +0.000, E1   -41.879, E3 +364667.275}
SPL {X  -159.484, Y  +684.213, Z    +0.000, E1   -41.818, E3 +364680.111}
SPL {X  -159.007, Y  +689.209, Z    +0.000, E1   -41.732, E3 +364692.416}
SPL {X  -158.327, Y  +694.511, Z    +0.000, E1   -41.622, E3 +364705.667}
SPL {X  -157.480, Y  +699.729, Z    +0.000, E1   -41.453, E3 +364718.930}
SPL {X  -156.604, Y  +704.242, Z    +0.000, E1   -41.288, E3 +364730.539}
SPL {X  -155.514, Y  +709.078, Z    +0.000, E1   -41.107, E3 +364743.093}
SPL {X  -154.232, Y  +714.035, Z    +0.000, E1   -40.861, E3 +364756.152}
SPL {X  -153.147, Y  +717.790, Z    +0.000, E1   -40.640, E3 +364766.170}
SPL {X  -151.881, Y  +721.788, Z    +0.000, E1   -40.435, E3 +364776.856}
SPL {X  -148.572, Y  +730.857, Z    +0.000, E1   -36.304, E3 +364833.065}
ENDSPLINE

SPLINE
SPL {X  -154.420, Y  +713.347, Z    +0.000, E1   -25.698, E3 +364878.489}
SPL {X  -156.970, Y  +702.437, Z    +0.000, E1   -20.224, E3 +364890.185}
SPL {X  -159.301, Y  +686.331, Z    +0.000, E1   -11.648, E3 +364899.958}
SPL {X  -159.936, Y  +675.651, Z    +0.000, E1    -5.377, E3 +364903.674}
SPL {X  -159.990, Y  +670.142, Z    +0.000, E1    -1.740, E3 +364904.974}
SPL {X  -159.990, Y  +666.629, Z    +0.000, E1    +0.827, E3 +364905.623}
SPL {X  -159.990, Y  +662.407, Z    +0.000, E1    +4.406, E3 +364906.473}
SPL {X  -159.990, Y  +655.884, Z    +0.000, E1   +10.601, E3 +364908.339}
SPL {X  -159.990, Y  +643.833, Z    +0.000, E1   +21.883, E3 +364913.968}
SPL {X  -159.990, Y  +617.235, Z    +0.000, E1   +36.481, E3 +364937.868}
SPL {X  -159.990, Y  +586.905, Z    +0.000, E1   +41.264, E3 +364986.845}
SPL {X  -159.990, Y  +581.111, Z    +0.000, E1   +41.245, E3 +365000.898}
SPL {X  -159.990, Y  +576.269, Z    +0.000, E1   +41.239, E3 +365012.626}
SPL {X  -159.990, Y  +571.714, Z    +0.000, E1   +41.240, E3 +365023.654}
SPL {X  -159.990, Y  +567.050, Z    +0.000, E1   +41.238, E3 +365034.941}
SPL {X  -159.990, Y  +561.959, Z    +0.000, E1   +41.251, E3 +365047.239}
SPL {X  -159.990, Y  +555.553, Z    +0.000, E1   +41.273, E3 +365062.707}
SPL {X  -159.990, Y  +549.897, Z    +0.000, E1   +41.240, E3 +365076.438}
SPL {X  -159.990, Y  +544.775, Z    +0.000, E1   +41.260, E3 +365088.812}
SPL {X  -159.990, Y  +538.952, Z    +0.000, E1   +41.247, E3 +365102.943}
SPL {X  -159.990, Y  +534.225, Z    +0.000, E1   +41.236, E3 +365114.377}
SPL {X  -159.990, Y  +529.136, Z    +0.000, E1   +41.262, E3 +365126.652}
SPL {X  -159.990, Y  +524.776, Z    +0.000, E1   +41.225, E3 +365137.266}
SPL {X  -159.990, Y  +521.454, Z    +0.000, E1   +41.236, E3 +365145.288}
SPL {X  -159.990, Y  +516.698, Z    +0.000, E1   +41.259, E3 +365156.727}
SPL {X  -159.990, Y  +510.896, Z    +0.000, E1   +41.267, E3 +365170.744}
SPL {X  -159.990, Y  +506.621, Z    +0.000, E1   +41.235, E3 +365181.146}
SPL {X  -159.990, Y  +501.314, Z    +0.000, E1   +41.284, E3 +365193.905}
SPL {X  -159.990, Y  +495.023, Z    +0.000, E1   +41.263, E3 +365209.136}
SPL {X  -159.990, Y  +479.011, Z    +0.000, E1   +45.740, E3 +365218.518}
SPL {X  -159.990, Y  +471.379, Z    +0.000, E1   +46.435, E3 +365230.134}
SPL {X  -159.990, Y  +465.881, Z    +0.000, E1   +45.385, E3 +365247.737}
SPL {X  -159.990, Y  +461.571, Z    +0.000, E1   +44.440, E3 +365262.262}
SPL {X  -159.990, Y  +458.229, Z    +0.000, E1   +43.579, E3 +365274.796}
SPL {X  -159.990, Y  +453.434, Z    +0.000, E1   +43.227, E3 +365287.570}
SPL {X  -159.990, Y  +448.702, Z    +0.000, E1   +43.218, E3 +365298.292}
SPL {X  -159.990, Y  +442.224, Z    +0.000, E1   +43.270, E3 +365312.842}
SPL {X  -159.990, Y  +434.411, Z    +0.000, E1   +43.246, E3 +365330.518}
SPL {X  -159.990, Y  +429.216, Z    +0.000, E1   +43.210, E3 +365342.291}
SPL {X  -159.990, Y  +424.433, Z    +0.000, E1   +43.237, E3 +365353.039}
SPL {X  -159.990, Y  +419.466, Z    +0.000, E1   +43.217, E3 +365364.278}
SPL {X  -159.990, Y  +414.585, Z    +0.000, E1   +43.233, E3 +365375.270}
SPL {X  -159.990, Y  +409.927, Z    +0.000, E1   +43.217, E3 +365385.802}
SPL {X  -159.990, Y  +405.428, Z    +0.000, E1   +43.230, E3 +365395.960}
SPL {X  -159.990, Y  +398.518, Z    +0.000, E1   +43.261, E3 +365411.514}
SPL {X  -159.990, Y  +392.163, Z    +0.000, E1   +43.223, E3 +365425.914}
SPL {X  -159.990, Y  +387.342, Z    +0.000, E1   +43.224, E3 +365436.792}
SPL {X  -159.990, Y  +382.548, Z    +0.000, E1   +43.224, E3 +365447.614}
SPL {X  -159.922, Y  +377.835, Z    +0.000, E1   +43.211, E3 +365458.331}
SPL {X  -159.608, Y  +371.448, Z    +0.000, E1   +43.200, E3 +365473.008}
SPL {X  -158.905, Y  +363.898, Z    +0.000, E1   +43.073, E3 +365490.776}
SPL {X  -158.182, Y  +358.518, Z    +0.000, E1   +42.902, E3 +365503.719}
SPL {X  -157.507, Y  +354.423, Z    +0.000, E1   +42.786, E3 +365513.665}
SPL {X  -156.676, Y  +350.104, Z    +0.000, E1   +42.637, E3 +365524.270}
SPL {X  -155.807, Y  +346.154, Z    +0.000, E1   +42.470, E3 +365534.097}
SPL {X  -154.777, Y  +341.993, Z    +0.000, E1   +42.302, E3 +365544.522}
SPL {X  -153.585, Y  +337.686, Z    +0.000, E1   +42.062, E3 +365555.498}
SPL {X  -152.412, Y  +333.846, Z    +0.000, E1   +41.856, E3 +365565.340}
SPL {X  -151.009, Y  +329.651, Z    +0.000, E1   +41.581, E3 +365576.240}
SPL {X  -148.356, Y  +322.607, Z    +0.000, E1   +36.121, E3 +365636.716}
ENDSPLINE

SPLINE
SPL {X  -156.487, Y  +349.204, Z    +0.000, E1   +21.338, E3 +365691.841}
SPL {X  -159.136, Y  +365.992, Z    +0.000, E1   +12.463, E3 +365702.600}
SPL {X  -159.799, Y  +374.694, Z    +0.000, E1    +7.504, E3 +365705.704}
SPL {X  -159.976, Y  +380.404, Z    +0.000, E1    +3.959, E3 +365707.237}
SPL {X  -159.990, Y  +384.773, Z    +0.000, E1    +1.003, E3 +365708.131}
SPL {X  -159.990, Y  +387.968, Z    +0.000, E1    -1.448, E3 +365708.700}
SPL {X  -159.990, Y  +391.397, Z    +0.000, E1    -4.422, E3 +365709.324}
SPL {X  -159.990, Y  +395.864, Z    +0.000, E1    -8.712, E3 +365710.412}
SPL {X  -159.990, Y  +401.273, Z    +0.000, E1   -14.176, E3 +365712.139}
SPL {X  -159.990, Y  +411.788, Z    +0.000, E1   -23.693, E3 +365717.682}
SPL {X  -159.990, Y  +438.158, Z    +0.000, E1   -37.630, E3 +365740.960}
SPL {X  -159.990, Y  +468.567, Z    +0.000, E1   -41.922, E3 +365790.303}
SPL {X  -159.990, Y  +474.616, Z    +0.000, E1   -41.909, E3 +365804.633}
SPL {X  -159.990, Y  +478.952, Z    +0.000, E1   -41.885, E3 +365814.931}
SPL {X  -159.990, Y  +484.724, Z    +0.000, E1   -41.943, E3 +365828.482}
SPL {X  -159.990, Y  +492.944, Z    +0.000, E1   -41.952, E3 +365847.902}
SPL {X  -159.990, Y  +499.538, Z    +0.000, E1   -41.904, E3 +365863.560}
SPL {X  -159.990, Y  +504.097, Z    +0.000, E1   -41.897, E3 +365874.349}
SPL {X  -159.990, Y  +509.413, Z    +0.000, E1   -41.921, E3 +365886.884}
SPL {X  -159.990, Y  +516.193, Z    +0.000, E1   -41.932, E3 +365902.900}
SPL {X  -159.990, Y  +521.318, Z    +0.000, E1   -41.891, E3 +365915.074}
SPL {X  -159.990, Y  +526.974, Z    +0.000, E1   -41.950, E3 +365928.364}
SPL {X  -159.990, Y  +533.758, Z    +0.000, E1   -41.910, E3 +365944.466}
SPL {X  -159.990, Y  +539.474, Z    +0.000, E1   -41.912, E3 +365957.994}
SPL {X  -159.990, Y  +544.879, Z    +0.000, E1   -41.899, E3 +365970.805}
SPL {X  -159.990, Y  +550.802, Z    +0.000, E1   -41.920, E3 +365984.786}
SPL {X  -159.990, Y  +556.952, Z    +0.000, E1   -41.911, E3 +365999.325}
SPL {X  -159.990, Y  +562.629, Z    +0.000, E1   -41.910, E3 +366012.744}
SPL {X  -159.990, Y  +567.682, Z    +0.000, E1   -41.901, E3 +366024.702}
SPL {X  -159.990, Y  +572.912, Z    +0.000, E1   -41.914, E3 +366037.050}
SPL {X  -159.990, Y  +578.863, Z    +0.000, E1   -41.918, E3 +366051.114}
SPL {X  -159.990, Y  +584.320, Z    +0.000, E1   -41.901, E3 +366064.061}
SPL {X  -159.990, Y  +589.217, Z    +0.000, E1   -41.901, E3 +366075.633}
SPL {X  -159.990, Y  +594.252, Z    +0.000, E1   -41.903, E3 +366087.548}
SPL {X  -159.990, Y  +600.237, Z    +0.000, E1   -41.928, E3 +366101.665}
SPL {X  -159.990, Y  +605.518, Z    +0.000, E1   -41.890, E3 +366114.203}
SPL {X  -159.990, Y  +610.545, Z    +0.000, E1   -41.917, E3 +366126.052}
SPL {X  -159.990, Y  +615.720, Z    +0.000, E1   -41.899, E3 +366138.312}
SPL {X  -159.990, Y  +621.417, Z    +0.000, E1   -41.931, E3 +366151.749}
SPL {X  -159.990, Y  +627.900, Z    +0.000, E1   -41.914, E3 +366167.088}
SPL {X  -159.990, Y  +632.270, Z    +0.000, E1   -41.887, E3 +366177.464}
SPL {X  -159.990, Y  +637.009, Z    +0.000, E1   -41.925, E3 +366188.607}
SPL {X  -159.990, Y  +642.624, Z    +0.000, E1   -41.901, E3 +366201.927}
SPL {X  -159.990, Y  +647.782, Z    +0.000, E1   -41.914, E3 +366214.096}
SPL {X  -159.990, Y  +653.094, Z    +0.000, E1   -41.905, E3 +366226.674}
SPL {X  -159.990, Y  +657.893, Z    +0.000, E1   -41.899, E3 +366238.040}
SPL {X  -159.990, Y  +662.516, Z    +0.000, E1   -41.899, E3 +366248.971}
SPL {X  -159.990, Y  +666.974, Z    +0.000, E1   -41.897, E3 +366259.515}
SPL {X  -159.984, Y  +672.859, Z    +0.000, E1   -41.934, E3 +366273.377}
SPL {X  -159.817, Y  +678.937, Z    +0.000, E1   -41.879, E3 +366287.965}
SPL {X  -159.484, Y  +684.213, Z    +0.000, E1   -41.818, E3 +366300.801}
SPL {X  -159.007, Y  +689.209, Z    +0.000, E1   -41.732, E3 +366313.106}
SPL {X  -158.327, Y  +694.511, Z    +0.000, E1   -41.622, E3 +366326.357}
SPL {X  -157.480, Y  +699.729, Z    +0.000, E1   -41.453, E3 +366339.620}
SPL {X  -156.604, Y  +704.242, Z    +0.000, E1   -41.288, E3 +366351.229}
SPL {X  -155.514, Y  +709.078, Z    +0.000, E1   -41.107, E3 +366363.782}
SPL {X  -154.232, Y  +714.035, Z    +0.000, E1   -40.861, E3 +366376.841}
SPL {X  -153.147, Y  +717.790, Z    +0.000, E1   -40.640, E3 +366386.859}
SPL {X  -151.881, Y  +721.788, Z    +0.000, E1   -40.435, E3 +366397.546}
SPL {X  -148.572, Y  +730.857, Z    +0.000, E1   -36.304, E3 +366453.755}
ENDSPLINE

SPLINE
SPL {X  -156.377, Y  +705.307, Z    +0.000, E1   -21.740, E3 +366508.004}
SPL {X  -158.965, Y  +689.585, Z    +0.000, E1   -13.405, E3 +366519.161}
SPL {X  -159.884, Y  +677.314, Z    +0.000, E1    -6.475, E3 +366523.874}
SPL {X  -159.990, Y  +670.142, Z    +0.000, E1    -1.740, E3 +366525.663}
SPL {X  -159.990, Y  +666.629, Z    +0.000, E1    +0.827, E3 +366526.313}
SPL {X  -159.990, Y  +662.407, Z    +0.000, E1    +4.406, E3 +366527.163}
SPL {X  -159.990, Y  +657.382, Z    +0.000, E1    +9.217, E3 +366528.545}
SPL {X  -159.990, Y  +653.255, Z    +0.000, E1   +13.347, E3 +366529.874}
SPL {X  -159.990, Y  +646.242, Z    +0.000, E1   +19.956, E3 +366532.948}
SPL {X  -159.990, Y  +624.365, Z    +0.000, E1   +33.860, E3 +366550.849}
SPL {X  -159.990, Y  +615.596, Z    +0.000, E1   +36.980, E3 +366560.508}
SPL {X  -159.990, Y  +586.905, Z    +0.000, E1   +41.264, E3 +366607.534}
SPL {X  -159.990, Y  +581.111, Z    +0.000, E1   +41.245, E3 +366621.588}
SPL {X  -159.990, Y  +576.269, Z    +0.000, E1   +41.239, E3 +366633.316}
SPL {X  -159.990, Y  +571.714, Z    +0.000, E1   +41.240, E3 +366644.344}
SPL {X  -159.990, Y  +567.050, Z    +0.000, E1   +41.238, E3 +366655.630}
SPL {X  -159.990, Y  +561.959, Z    +0.000, E1   +41.251, E3 +366667.929}
SPL {X  -159.990, Y  +555.553, Z    +0.000, E1   +41.273, E3 +366683.397}
SPL {X  -159.990, Y  +549.897, Z    +0.000, E1   +41.240, E3 +366697.127}
SPL {X  -159.990, Y  +544.775, Z    +0.000, E1   +41.260, E3 +366709.502}
SPL {X  -159.990, Y  +538.952, Z    +0.000, E1   +41.247, E3 +366723.633}
SPL {X  -159.990, Y  +534.225, Z    +0.000, E1   +41.236, E3 +366735.066}
SPL {X  -159.990, Y  +529.136, Z    +0.000, E1   +41.262, E3 +366747.342}
SPL {X  -159.990, Y  +524.776, Z    +0.000, E1   +41.225, E3 +366757.956}
SPL {X  -159.990, Y  +521.454, Z    +0.000, E1   +41.236, E3 +366765.977}
SPL {X  -159.990, Y  +515.605, Z    +0.000, E1   +41.288, E3 +366780.017}
SPL {X  -159.990, Y  +509.898, Z    +0.000, E1   +41.246, E3 +366793.878}
SPL {X  -159.990, Y  +505.215, Z    +0.000, E1   +41.261, E3 +366805.194}
SPL {X  -159.990, Y  +498.837, Z    +0.000, E1   +41.283, E3 +366820.582}
SPL {X  -159.990, Y  +493.848, Z    +0.000, E1   +41.241, E3 +366832.702}
SPL {X  -159.990, Y  +479.011, Z    +0.000, E1   +45.740, E3 +366839.208}
SPL {X  -159.990, Y  +471.379, Z    +0.000, E1   +46.435, E3 +366850.823}
SPL {X  -159.990, Y  +466.895, Z    +0.000, E1   +45.533, E3 +366865.228}
SPL {X  -159.990, Y  +462.409, Z    +0.000, E1   +44.664, E3 +366880.003}
SPL {X  -159.990, Y  +458.229, Z    +0.000, E1   +43.579, E3 +366895.485}
SPL {X  -159.990, Y  +453.434, Z    +0.000, E1   +43.227, E3 +366908.260}
SPL {X  -159.990, Y  +448.702, Z    +0.000, E1   +43.218, E3 +366918.982}
SPL {X  -159.990, Y  +444.476, Z    +0.000, E1   +43.219, E3 +366928.520}
SPL {X  -159.990, Y  +440.246, Z    +0.000, E1   +43.217, E3 +366938.078}
SPL {X  -159.990, Y  +434.411, Z    +0.000, E1   +43.246, E3 +366951.208}
SPL {X  -159.990, Y  +429.216, Z    +0.000, E1   +43.210, E3 +366962.980}
SPL {X  -159.990, Y  +424.433, Z    +0.000, E1   +43.237, E3 +366973.728}
SPL {X  -159.990, Y  +419.466, Z    +0.000, E1   +43.217, E3 +366984.968}
SPL {X  -159.990, Y  +414.585, Z    +0.000, E1   +43.233, E3 +366995.960}
SPL {X  -159.990, Y  +409.927, Z    +0.000, E1   +43.217, E3 +367006.491}
SPL {X  -159.990, Y  +405.428, Z    +0.000, E1   +43.230, E3 +367016.650}
SPL {X  -159.990, Y  +401.033, Z    +0.000, E1   +43.209, E3 +367026.604}
SPL {X  -159.990, Y  +396.968, Z    +0.000, E1   +43.221, E3 +367035.762}
SPL {X  -159.990, Y  +392.163, Z    +0.000, E1   +43.223, E3 +367046.604}
SPL {X  -159.990, Y  +387.342, Z    +0.000, E1   +43.224, E3 +367057.481}
SPL {X  -159.990, Y  +382.548, Z    +0.000, E1   +43.224, E3 +367068.304}
SPL {X  -159.922, Y  +377.835, Z    +0.000, E1   +43.211, E3 +367079.021}
SPL {X  -159.712, Y  +373.072, Z    +0.000, E1   +43.177, E3 +367089.987}
SPL {X  -159.289, Y  +367.537, Z    +0.000, E1   +43.118, E3 +367102.899}
SPL {X  -158.730, Y  +362.464, Z    +0.000, E1   +43.003, E3 +367114.931}
SPL {X  -158.182, Y  +358.518, Z    +0.000, E1   +42.902, E3 +367124.409}
SPL {X  -157.507, Y  +354.423, Z    +0.000, E1   +42.786, E3 +367134.354}
SPL {X  -156.676, Y  +350.104, Z    +0.000, E1   +42.637, E3 +367144.960}
SPL {X  -155.807, Y  +346.154, Z    +0.000, E1   +42.470, E3 +367154.787}
SPL {X  -154.777, Y  +341.993, Z    +0.000, E1   +42.302, E3 +367165.212}
SPL {X  -153.585, Y  +337.686, Z    +0.000, E1   +42.062, E3 +367176.187}
SPL {X  -152.412, Y  +333.846, Z    +0.000, E1   +41.856, E3 +367186.030}
SPL {X  -151.009, Y  +329.651, Z    +0.000, E1   +41.581, E3 +367196.930}
SPL {X  -148.356, Y  +322.607, Z    +0.000, E1   +36.121, E3 +367257.405}
ENDSPLINE

SPLINE
SPL {X  -156.487, Y  +349.204, Z    +0.000, E1   +21.338, E3 +367312.531}
SPL {X  -159.136, Y  +365.992, Z    +0.000, E1   +12.463, E3 +367323.290}
SPL {X  -159.799, Y  +374.694, Z    +0.000, E1    +7.504, E3 +367326.393}
SPL {X  -159.976, Y  +380.404, Z    +0.000, E1    +3.959, E3 +367327.926}
SPL {X  -159.990, Y  +384.773, Z    +0.000, E1    +1.003, E3 +367328.821}
SPL {X  -159.990, Y  +387.968, Z    +0.000, E1    -1.448, E3 +367329.389}
SPL {X  -159.990, Y  +391.397, Z    +0.000, E1    -4.422, E3 +367330.013}
SPL {X  -159.990, Y  +395.864, Z    +0.000, E1    -8.712, E3 +367331.102}
SPL {X  -159.990, Y  +401.273, Z    +0.000, E1   -14.176, E3 +367332.829}
SPL {X  -159.990, Y  +411.788, Z    +0.000, E1   -23.693, E3 +367338.372}
SPL {X  -159.990, Y  +438.158, Z    +0.000, E1   -37.630, E3 +367361.649}
SPL {X  -159.990, Y  +468.567, Z    +0.000, E1   -41.922, E3 +367410.993}
SPL {X  -159.990, Y  +474.616, Z    +0.000, E1   -41.909, E3 +367425.323}
SPL {X  -159.990, Y  +478.952, Z    +0.000, E1   -41.885, E3 +367435.620}
SPL {X  -159.990, Y  +484.724, Z    +0.000, E1   -41.943, E3 +367449.172}
SPL {X  -159.990, Y  +492.944, Z    +0.000, E1   -41.952, E3 +367468.592}
SPL {X  -159.990, Y  +499.538, Z    +0.000, E1   -41.904, E3 +367484.250}
SPL {X  -159.990, Y  +504.097, Z    +0.000, E1   -41.897, E3 +367495.039}
SPL {X  -159.990, Y  +509.413, Z    +0.000, E1   -41.921, E3 +367507.574}
SPL {X  -159.990, Y  +516.193, Z    +0.000, E1   -41.932, E3 +367523.590}
SPL {X  -159.990, Y  +521.318, Z    +0.000, E1   -41.891, E3 +367535.764}
SPL {X  -159.990, Y  +526.974, Z    +0.000, E1   -41.950, E3 +367549.053}
SPL {X  -159.990, Y  +533.758, Z    +0.000, E1   -41.910, E3 +367565.156}
SPL {X  -159.990, Y  +539.474, Z    +0.000, E1   -41.912, E3 +367578.683}
SPL {X  -159.990, Y  +544.879, Z    +0.000, E1   -41.899, E3 +367591.495}
SPL {X  -159.990, Y  +550.802, Z    +0.000, E1   -41.920, E3 +367605.476}
SPL {X  -159.990, Y  +556.952, Z    +0.000, E1   -41.911, E3 +367620.015}
SPL {X  -159.990, Y  +562.629, Z    +0.000, E1   -41.910, E3 +367633.433}
SPL {X  -159.990, Y  +567.682, Z    +0.000, E1   -41.901, E3 +367645.392}
SPL {X  -159.990, Y  +572.912, Z    +0.000, E1   -41.914, E3 +367657.739}
SPL {X  -159.990, Y  +578.863, Z    +0.000, E1   -41.918, E3 +367671.803}
SPL {X  -159.990, Y  +584.320, Z    +0.000, E1   -41.901, E3 +367684.750}
SPL {X  -159.990, Y  +589.217, Z    +0.000, E1   -41.901, E3 +367696.323}
SPL {X  -159.990, Y  +594.252, Z    +0.000, E1   -41.903, E3 +367708.238}
SPL {X  -159.990, Y  +600.237, Z    +0.000, E1   -41.928, E3 +367722.355}
SPL {X  -159.990, Y  +605.518, Z    +0.000, E1   -41.890, E3 +367734.893}
SPL {X  -159.990, Y  +610.545, Z    +0.000, E1   -41.917, E3 +367746.741}
SPL {X  -159.990, Y  +615.720, Z    +0.000, E1   -41.899, E3 +367759.002}
SPL {X  -159.990, Y  +621.417, Z    +0.000, E1   -41.931, E3 +367772.438}
SPL {X  -159.990, Y  +627.900, Z    +0.000, E1   -41.914, E3 +367787.778}
SPL {X  -159.990, Y  +632.270, Z    +0.000, E1   -41.887, E3 +367798.154}
SPL {X  -159.990, Y  +637.009, Z    +0.000, E1   -41.925, E3 +367809.296}
SPL {X  -159.990, Y  +642.624, Z    +0.000, E1   -41.901, E3 +367822.617}
SPL {X  -159.990, Y  +647.782, Z    +0.000, E1   -41.914, E3 +367834.786}
SPL {X  -159.990, Y  +653.094, Z    +0.000, E1   -41.905, E3 +367847.364}
SPL {X  -159.990, Y  +657.893, Z    +0.000, E1   -41.899, E3 +367858.729}
SPL {X  -159.990, Y  +662.516, Z    +0.000, E1   -41.899, E3 +367869.661}
SPL {X  -159.990, Y  +666.974, Z    +0.000, E1   -41.897, E3 +367880.205}
SPL {X  -159.984, Y  +672.859, Z    +0.000, E1   -41.934, E3 +367894.066}
SPL {X  -159.817, Y  +678.937, Z    +0.000, E1   -41.879, E3 +367908.655}
SPL {X  -159.484, Y  +684.213, Z    +0.000, E1   -41.818, E3 +367921.491}
SPL {X  -159.007, Y  +689.209, Z    +0.000, E1   -41.732, E3 +367933.796}
SPL {X  -158.327, Y  +694.511, Z    +0.000, E1   -41.622, E3 +367947.047}
SPL {X  -157.480, Y  +699.729, Z    +0.000, E1   -41.453, E3 +367960.309}
SPL {X  -156.604, Y  +704.242, Z    +0.000, E1   -41.288, E3 +367971.918}
SPL {X  -155.514, Y  +709.078, Z    +0.000, E1   -41.107, E3 +367984.472}
SPL {X  -154.232, Y  +714.035, Z    +0.000, E1   -40.861, E3 +367997.531}
SPL {X  -153.147, Y  +717.790, Z    +0.000, E1   -40.640, E3 +368007.549}
SPL {X  -151.881, Y  +721.788, Z    +0.000, E1   -40.435, E3 +368018.236}
SPL {X  -148.572, Y  +730.857, Z    +0.000, E1   -36.304, E3 +368074.445}
ENDSPLINE

SPLINE
SPL {X  -156.377, Y  +705.307, Z    +0.000, E1   -21.740, E3 +368128.693}
SPL {X  -158.965, Y  +689.585, Z    +0.000, E1   -13.405, E3 +368139.851}
SPL {X  -159.884, Y  +677.314, Z    +0.000, E1    -6.475, E3 +368144.564}
SPL {X  -159.990, Y  +670.142, Z    +0.000, E1    -1.740, E3 +368146.353}
SPL {X  -159.990, Y  +666.629, Z    +0.000, E1    +0.827, E3 +368147.002}
SPL {X  -159.990, Y  +662.407, Z    +0.000, E1    +4.406, E3 +368147.853}
SPL {X  -159.990, Y  +655.884, Z    +0.000, E1   +10.601, E3 +368149.718}
SPL {X  -159.990, Y  +643.833, Z    +0.000, E1   +21.883, E3 +368155.347}
SPL {X  -159.990, Y  +617.235, Z    +0.000, E1   +36.481, E3 +368179.247}
SPL {X  -159.990, Y  +586.905, Z    +0.000, E1   +41.264, E3 +368228.224}
SPL {X  -159.990, Y  +581.111, Z    +0.000, E1   +41.245, E3 +368242.278}
SPL {X  -159.990, Y  +576.269, Z    +0.000, E1   +41.239, E3 +368254.005}
SPL {X  -159.990, Y  +571.714, Z    +0.000, E1   +41.240, E3 +368265.033}
SPL {X  -159.990, Y  +567.050, Z    +0.000, E1   +41.238, E3 +368276.320}
SPL {X  -159.990, Y  +561.959, Z    +0.000, E1   +41.251, E3 +368288.619}
SPL {X  -159.990, Y  +555.553, Z    +0.000, E1   +41.273, E3 +368304.087}
SPL {X  -159.990, Y  +549.897, Z    +0.000, E1   +41.240, E3 +368317.817}
SPL {X  -159.990, Y  +544.775, Z    +0.000, E1   +41.260, E3 +368330.192}
SPL {X  -159.990, Y  +540.176, Z    +0.000, E1   +41.224, E3 +368341.401}
SPL {X  -159.990, Y  +534.009, Z    +0.000, E1   +41.300, E3 +368356.186}
SPL {X  -159.990, Y  +526.579, Z    +0.000, E1   +41.262, E3 +368374.223}
SPL {X  -159.990, Y  +521.454, Z    +0.000, E1   +41.236, E3 +368386.667}
SPL {X  -159.990, Y  +516.698, Z    +0.000, E1   +41.259, E3 +368398.106}
SPL {X  -159.990, Y  +510.896, Z    +0.000, E1   +41.267, E3 +368412.124}
SPL {X  -159.990, Y  +505.215, Z    +0.000, E1   +41.261, E3 +368425.884}
SPL {X  -159.990, Y  +500.102, Z    +0.000, E1   +41.251, E3 +368438.267}
SPL {X  -159.990, Y  +495.023, Z    +0.000, E1   +41.263, E3 +368450.516}
SPL {X  -159.990, Y  +479.011, Z    +0.000, E1   +45.740, E3 +368459.898}
SPL {X  -159.990, Y  +471.379, Z    +0.000, E1   +46.435, E3 +368471.513}
SPL {X  -159.990, Y  +466.895, Z    +0.000, E1   +45.533, E3 +368485.918}
SPL {X  -159.990, Y  +462.409, Z    +0.000, E1   +44.664, E3 +368500.693}
SPL {X  -159.990, Y  +458.229, Z    +0.000, E1   +43.579, E3 +368516.175}
SPL {X  -159.990, Y  +453.434, Z    +0.000, E1   +43.227, E3 +368528.949}
SPL {X  -159.990, Y  +448.702, Z    +0.000, E1   +43.218, E3 +368539.671}
SPL {X  -159.990, Y  +444.476, Z    +0.000, E1   +43.219, E3 +368549.210}
SPL {X  -159.990, Y  +440.246, Z    +0.000, E1   +43.217, E3 +368558.767}
SPL {X  -159.990, Y  +434.411, Z    +0.000, E1   +43.246, E3 +368571.897}
SPL {X  -159.990, Y  +429.216, Z    +0.000, E1   +43.210, E3 +368583.670}
SPL {X  -159.990, Y  +424.433, Z    +0.000, E1   +43.237, E3 +368594.418}
SPL {X  -159.990, Y  +419.466, Z    +0.000, E1   +43.217, E3 +368605.657}
SPL {X  -159.990, Y  +414.585, Z    +0.000, E1   +43.233, E3 +368616.649}
SPL {X  -159.990, Y  +409.927, Z    +0.000, E1   +43.217, E3 +368627.181}
SPL {X  -159.990, Y  +405.428, Z    +0.000, E1   +43.230, E3 +368637.339}
SPL {X  -159.990, Y  +398.518, Z    +0.000, E1   +43.261, E3 +368652.894}
SPL {X  -159.990, Y  +392.163, Z    +0.000, E1   +43.223, E3 +368667.294}
SPL {X  -159.990, Y  +387.342, Z    +0.000, E1   +43.224, E3 +368678.171}
SPL {X  -159.990, Y  +382.548, Z    +0.000, E1   +43.224, E3 +368688.994}
SPL {X  -159.922, Y  +377.835, Z    +0.000, E1   +43.211, E3 +368699.711}
SPL {X  -159.712, Y  +373.072, Z    +0.000, E1   +43.177, E3 +368710.677}
SPL {X  -159.289, Y  +367.537, Z    +0.000, E1   +43.118, E3 +368723.588}
SPL {X  -158.730, Y  +362.464, Z    +0.000, E1   +43.003, E3 +368735.620}
SPL {X  -158.182, Y  +358.518, Z    +0.000, E1   +42.902, E3 +368745.099}
SPL {X  -157.507, Y  +354.423, Z    +0.000, E1   +42.786, E3 +368755.044}
SPL {X  -156.676, Y  +350.104, Z    +0.000, E1   +42.637, E3 +368765.649}
SPL {X  -155.807, Y  +346.154, Z    +0.000, E1   +42.470, E3 +368775.476}
SPL {X  -154.777, Y  +341.993, Z    +0.000, E1   +42.302, E3 +368785.902}
SPL {X  -153.585, Y  +337.686, Z    +0.000, E1   +42.062, E3 +368796.877}
SPL {X  -152.412, Y  +333.846, Z    +0.000, E1   +41.856, E3 +368806.720}
SPL {X  -151.009, Y  +329.651, Z    +0.000, E1   +41.581, E3 +368817.619}
SPL {X  -148.356, Y  +322.607, Z    +0.000, E1   +36.121, E3 +368878.095}
ENDSPLINE

SPLINE
SPL {X  -156.487, Y  +349.204, Z    +0.000, E1   +21.338, E3 +368933.221}
SPL {X  -159.136, Y  +365.992, Z    +0.000, E1   +12.463, E3 +368943.979}
SPL {X  -159.799, Y  +374.694, Z    +0.000, E1    +7.504, E3 +368947.083}
SPL {X  -159.976, Y  +380.404, Z    +0.000, E1    +3.959, E3 +368948.616}
SPL {X  -159.990, Y  +384.773, Z    +0.000, E1    +1.003, E3 +368949.511}
SPL {X  -159.990, Y  +387.968, Z    +0.000, E1    -1.448, E3 +368950.079}
SPL {X  -159.990, Y  +391.397, Z    +0.000, E1    -4.422, E3 +368950.703}
SPL {X  -159.990, Y  +395.864, Z    +0.000, E1    -8.712, E3 +368951.791}
SPL {X  -159.990, Y  +401.273, Z    +0.000, E1   -14.176, E3 +368953.519}
SPL {X  -159.990, Y  +409.369, Z    +0.000, E1   -21.807, E3 +368957.311}
SPL {X  -159.990, Y  +436.107, Z    +0.000, E1   -36.921, E3 +368980.236}
SPL {X  -159.990, Y  +468.567, Z    +0.000, E1   -41.922, E3 +369031.683}
SPL {X  -159.990, Y  +474.616, Z    +0.000, E1   -41.909, E3 +369046.012}
SPL {X  -159.990, Y  +478.952, Z    +0.000, E1   -41.885, E3 +369056.310}
SPL {X  -159.990, Y  +484.724, Z    +0.000, E1   -41.943, E3 +369069.862}
SPL {X  -159.990, Y  +492.944, Z    +0.000, E1   -41.952, E3 +369089.281}
SPL {X  -159.990, Y  +499.538, Z    +0.000, E1   -41.904, E3 +369104.940}
SPL {X  -159.990, Y  +504.097, Z    +0.000, E1   -41.897, E3 +369115.728}
SPL {X  -159.990, Y  +509.413, Z    +0.000, E1   -41.921, E3 +369128.263}
SPL {X  -159.990, Y  +516.193, Z    +0.000, E1   -41.932, E3 +369144.280}
SPL {X  -159.990, Y  +523.027, Z    +0.000, E1   -41.926, E3 +369160.441}
SPL {X  -159.990, Y  +528.611, Z    +0.000, E1   -41.900, E3 +369173.696}
SPL {X  -159.990, Y  +533.758, Z    +0.000, E1   -41.910, E3 +369185.845}
SPL {X  -159.990, Y  +539.474, Z    +0.000, E1   -41.912, E3 +369199.373}
SPL {X  -159.990, Y  +544.879, Z    +0.000, E1   -41.899, E3 +369212.184}
SPL {X  -159.990, Y  +550.802, Z    +0.000, E1   -41.920, E3 +369226.166}
SPL {X  -159.990, Y  +556.952, Z    +0.000, E1   -41.911, E3 +369240.705}
SPL {X  -159.990, Y  +562.629, Z    +0.000, E1   -41.910, E3 +369254.123}
SPL {X  -159.990, Y  +567.682, Z    +0.000, E1   -41.901, E3 +369266.082}
SPL {X  -159.990, Y  +574.350, Z    +0.000, E1   -41.955, E3 +369281.767}
SPL {X  -159.990, Y  +580.118, Z    +0.000, E1   -41.891, E3 +369295.504}
SPL {X  -159.990, Y  +584.320, Z    +0.000, E1   -41.901, E3 +369305.440}
SPL {X  -159.990, Y  +589.217, Z    +0.000, E1   -41.901, E3 +369317.013}
SPL {X  -159.990, Y  +594.252, Z    +0.000, E1   -41.903, E3 +369328.927}
SPL {X  -159.990, Y  +600.237, Z    +0.000, E1   -41.928, E3 +369343.045}
SPL {X  -159.990, Y  +605.518, Z    +0.000, E1   -41.890, E3 +369355.583}
SPL {X  -159.990, Y  +610.545, Z    +0.000, E1   -41.917, E3 +369367.431}
SPL {X  -159.990, Y  +615.720, Z    +0.000, E1   -41.899, E3 +369379.691}
SPL {X  -159.990, Y  +620.005, Z    +0.000, E1   -41.900, E3 +369389.824}
SPL {X  -159.990, Y  +624.919, Z    +0.000, E1   -41.912, E3 +369401.432}
SPL {X  -159.990, Y  +629.282, Z    +0.000, E1   -41.888, E3 +369411.772}
SPL {X  -159.990, Y  +634.411, Z    +0.000, E1   -41.931, E3 +369423.837}
SPL {X  -159.990, Y  +641.479, Z    +0.000, E1   -41.931, E3 +369440.553}
SPL {X  -159.990, Y  +647.782, Z    +0.000, E1   -41.914, E3 +369455.475}
SPL {X  -159.990, Y  +653.094, Z    +0.000, E1   -41.905, E3 +369468.054}
SPL {X  -159.990, Y  +657.893, Z    +0.000, E1   -41.899, E3 +369479.419}
SPL {X  -159.990, Y  +662.516, Z    +0.000, E1   -41.899, E3 +369490.350}
SPL {X  -159.990, Y  +668.411, Z    +0.000, E1   -41.929, E3 +369504.244}
SPL {X  -159.968, Y  +674.139, Z    +0.000, E1   -41.898, E3 +369517.848}
SPL {X  -159.817, Y  +678.937, Z    +0.000, E1   -41.879, E3 +369529.344}
SPL {X  -159.484, Y  +684.213, Z    +0.000, E1   -41.818, E3 +369542.180}
SPL {X  -159.007, Y  +689.209, Z    +0.000, E1   -41.732, E3 +369554.485}
SPL {X  -158.327, Y  +694.511, Z    +0.000, E1   -41.622, E3 +369567.736}
SPL {X  -157.480, Y  +699.729, Z    +0.000, E1   -41.453, E3 +369580.999}
SPL {X  -156.604, Y  +704.242, Z    +0.000, E1   -41.288, E3 +369592.608}
SPL {X  -155.831, Y  +707.744, Z    +0.000, E1   -41.132, E3 +369601.728}
SPL {X  -155.167, Y  +710.488, Z    +0.000, E1   -41.008, E3 +369608.906}
SPL {X  -154.232, Y  +714.035, Z    +0.000, E1   -40.861, E3 +369618.221}
SPL {X  -153.147, Y  +717.790, Z    +0.000, E1   -40.640, E3 +369628.239}
SPL {X  -151.881, Y  +721.788, Z    +0.000, E1   -40.435, E3 +369638.925}
SPL {X  -148.572, Y  +730.857, Z    +0.000, E1   -36.304, E3 +369695.134}
ENDSPLINE

SPLINE
SPL {X  -156.377, Y  +705.307, Z    +0.000, E1   -21.740, E3 +369749.383}
SPL {X  -159.301, Y  +686.331, Z    +0.000, E1   -11.648, E3 +369762.027}
SPL {X  -159.936, Y  +675.651, Z    +0.000, E1    -5.377, E3 +369765.743}
SPL {X  -159.990, Y  +670.142, Z    +0.000, E1    -1.740, E3 +369767.043}
SPL {X  -159.990, Y  +666.629, Z    +0.000, E1    +0.827, E3 +369767.692}
SPL {X  -159.990, Y  +662.407, Z    +0.000, E1    +4.406, E3 +369768.542}
SPL {X  -159.990, Y  +655.884, Z    +0.000, E1   +10.601, E3 +369770.408}
SPL {X  -159.990, Y  +643.833, Z    +0.000, E1   +21.883, E3 +369776.037}
SPL {X  -159.990, Y  +617.235, Z    +0.000, E1   +36.481, E3 +369799.937}
SPL {X  -159.990, Y  +586.905, Z    +0.000, E1   +41.264, E3 +369848.913}
SPL {X  -159.990, Y  +581.111, Z    +0.000, E1   +41.245, E3 +369862.967}
SPL {X  -159.990, Y  +576.269, Z    +0.000, E1   +41.239, E3 +369874.695}
SPL {X  -159.990, Y  +571.714, Z    +0.000, E1   +41.240, E3 +369885.723}
SPL {X  -159.990, Y  +567.050, Z    +0.000, E1   +41.238, E3 +369897.010}
SPL {X  -159.990, Y  +561.959, Z    +0.000, E1   +41.251, E3 +369909.308}
SPL {X  -159.990, Y  +555.553, Z    +0.000, E1   +41.273, E3 +369924.776}
SPL {X  -159.990, Y  +549.897, Z    +0.000, E1   +41.240, E3 +369938.507}
SPL {X  -159.990, Y  +544.775, Z    +0.000, E1   +41.260, E3 +369950.881}
SPL {X  -159.990, Y  +538.952, Z    +0.000, E1   +41.247, E3 +369965.012}
SPL {X  -159.990, Y  +534.225, Z    +0.000, E1   +41.236, E3 +369976.446}
SPL {X  -159.990, Y  +529.136, Z    +0.000, E1   +41.262, E3 +369988.721}
SPL {X  -159.990, Y  +522.690, Z    +0.000, E1   +41.265, E3 +370004.321}
SPL {X  -159.990, Y  +516.698, Z    +0.000, E1   +41.259, E3 +370018.795}
SPL {X  -159.990, Y  +510.896, Z    +0.000, E1   +41.267, E3 +370032.813}
SPL {X  -159.990, Y  +505.215, Z    +0.000, E1   +41.261, E3 +370046.573}
SPL {X  -159.990, Y  +500.102, Z    +0.000, E1   +41.251, E3 +370058.956}
SPL {X  -159.990, Y  +495.023, Z    +0.000, E1   +41.263, E3 +370071.205}
SPL {X  -159.990, Y  +479.011, Z    +0.000, E1   +45.740, E3 +370080.587}
SPL {X  -159.990, Y  +471.379, Z    +0.000, E1   +46.435, E3 +370092.203}
SPL {X  -159.990, Y  +465.881, Z    +0.000, E1   +45.385, E3 +370109.806}
SPL {X  -159.990, Y  +461.571, Z    +0.000, E1   +44.440, E3 +370124.331}
SPL {X  -159.990, Y  +458.229, Z    +0.000, E1   +43.579, E3 +370136.865}
SPL {X  -159.990, Y  +453.434, Z    +0.000, E1   +43.227, E3 +370149.639}
SPL {X  -159.990, Y  +448.702, Z    +0.000, E1   +43.218, E3 +370160.361}
SPL {X  -159.990, Y  +444.476, Z    +0.000, E1   +43.219, E3 +370169.899}
SPL {X  -159.990, Y  +440.246, Z    +0.000, E1   +43.217, E3 +370179.457}
SPL {X  -159.990, Y  +434.411, Z    +0.000, E1   +43.246, E3 +370192.587}
SPL {X  -159.990, Y  +429.216, Z    +0.000, E1   +43.210, E3 +370204.360}
SPL {X  -159.990, Y  +424.433, Z    +0.000, E1   +43.237, E3 +370215.108}
SPL {X  -159.990, Y  +419.466, Z    +0.000, E1   +43.217, E3 +370226.347}
SPL {X  -159.990, Y  +414.585, Z    +0.000, E1   +43.233, E3 +370237.339}
SPL {X  -159.990, Y  +409.927, Z    +0.000, E1   +43.217, E3 +370247.871}
SPL {X  -159.990, Y  +405.428, Z    +0.000, E1   +43.230, E3 +370258.029}
SPL {X  -159.990, Y  +398.518, Z    +0.000, E1   +43.261, E3 +370273.583}
SPL {X  -159.990, Y  +392.163, Z    +0.000, E1   +43.223, E3 +370287.983}
SPL {X  -159.990, Y  +387.342, Z    +0.000, E1   +43.224, E3 +370298.861}
SPL {X  -159.990, Y  +382.548, Z    +0.000, E1   +43.224, E3 +370309.683}
SPL {X  -159.922, Y  +377.835, Z    +0.000, E1   +43.211, E3 +370320.400}
SPL {X  -159.712, Y  +373.072, Z    +0.000, E1   +43.177, E3 +370331.366}
SPL {X  -159.289, Y  +367.537, Z    +0.000, E1   +43.118, E3 +370344.278}
SPL {X  -158.730, Y  +362.464, Z    +0.000, E1   +43.003, E3 +370356.310}
SPL {X  -158.182, Y  +358.518, Z    +0.000, E1   +42.902, E3 +370365.788}
SPL {X  -157.507, Y  +354.423, Z    +0.000, E1   +42.786, E3 +370375.734}
SPL {X  -156.676, Y  +350.104, Z    +0.000, E1   +42.637, E3 +370386.339}
SPL {X  -155.807, Y  +346.154, Z    +0.000, E1   +42.470, E3 +370396.166}
SPL {X  -154.777, Y  +341.993, Z    +0.000, E1   +42.302, E3 +370406.591}
SPL {X  -153.585, Y  +337.686, Z    +0.000, E1   +42.062, E3 +370417.567}
SPL {X  -152.412, Y  +333.846, Z    +0.000, E1   +41.856, E3 +370427.409}
SPL {X  -151.009, Y  +329.651, Z    +0.000, E1   +41.581, E3 +370438.309}
SPL {X  -148.356, Y  +322.607, Z    +0.000, E1   +36.121, E3 +370498.785}
ENDSPLINE

SPLINE
SPL {X  -156.487, Y  +349.204, Z    +0.000, E1   +21.338, E3 +370553.910}
SPL {X  -159.136, Y  +365.992, Z    +0.000, E1   +12.463, E3 +370564.669}
SPL {X  -159.799, Y  +374.694, Z    +0.000, E1    +7.504, E3 +370567.773}
SPL {X  -159.976, Y  +380.404, Z    +0.000, E1    +3.959, E3 +370569.306}
SPL {X  -159.990, Y  +384.773, Z    +0.000, E1    +1.003, E3 +370570.200}
SPL {X  -159.990, Y  +387.968, Z    +0.000, E1    -1.448, E3 +370570.769}
SPL {X  -159.990, Y  +391.397, Z    +0.000, E1    -4.422, E3 +370571.393}
SPL {X  -159.990, Y  +395.864, Z    +0.000, E1    -8.712, E3 +370572.481}
SPL {X  -159.990, Y  +401.273, Z    +0.000, E1   -14.176, E3 +370574.208}
SPL {X  -159.990, Y  +409.369, Z    +0.000, E1   -21.807, E3 +370578.000}
SPL {X  -159.990, Y  +436.107, Z    +0.000, E1   -36.921, E3 +370600.925}
SPL {X  -159.990, Y  +469.969, Z    +0.000, E1   -41.961, E3 +370655.630}
SPL {X  -159.990, Y  +477.498, Z    +0.000, E1   -41.916, E3 +370673.513}
SPL {X  -159.990, Y  +483.140, Z    +0.000, E1   -41.902, E3 +370686.869}
SPL {X  -159.990, Y  +488.618, Z    +0.000, E1   -41.913, E3 +370699.801}
SPL {X  -159.990, Y  +494.299, Z    +0.000, E1   -41.910, E3 +370713.235}
SPL {X  -159.990, Y  +499.538, Z    +0.000, E1   -41.904, E3 +370725.629}
SPL {X  -159.990, Y  +504.097, Z    +0.000, E1   -41.897, E3 +370736.418}
SPL {X  -159.990, Y  +509.413, Z    +0.000, E1   -41.921, E3 +370748.953}
SPL {X  -159.990, Y  +513.834, Z    +0.000, E1   -41.885, E3 +370759.466}
SPL {X  -159.990, Y  +517.450, Z    +0.000, E1   -41.901, E3 +370767.986}
SPL {X  -159.990, Y  +523.027, Z    +0.000, E1   -41.926, E3 +370781.131}
SPL {X  -159.990, Y  +528.611, Z    +0.000, E1   -41.900, E3 +370794.386}
SPL {X  -159.990, Y  +533.758, Z    +0.000, E1   -41.910, E3 +370806.535}
SPL {X  -159.990, Y  +539.474, Z    +0.000, E1   -41.912, E3 +370820.062}
SPL {X  -159.990, Y  +544.879, Z    +0.000, E1   -41.899, E3 +370832.874}
SPL {X  -159.990, Y  +550.802, Z    +0.000, E1   -41.920, E3 +370846.855}
SPL {X  -159.990, Y  +556.952, Z    +0.000, E1   -41.911, E3 +370861.394}
SPL {X  -159.990, Y  +562.629, Z    +0.000, E1   -41.910, E3 +370874.812}
SPL {X  -159.990, Y  +567.682, Z    +0.000, E1   -41.901, E3 +370886.771}
SPL {X  -159.990, Y  +572.912, Z    +0.000, E1   -41.914, E3 +370899.119}
SPL {X  -159.990, Y  +578.863, Z    +0.000, E1   -41.918, E3 +370913.183}
SPL {X  -159.990, Y  +584.320, Z    +0.000, E1   -41.901, E3 +370926.129}
SPL {X  -159.990, Y  +589.217, Z    +0.000, E1   -41.901, E3 +370937.702}
SPL {X  -159.990, Y  +594.252, Z    +0.000, E1   -41.903, E3 +370949.617}
SPL {X  -159.990, Y  +598.793, Z    +0.000, E1   -41.896, E3 +370960.371}
SPL {X  -159.990, Y  +604.215, Z    +0.000, E1   -41.919, E3 +370973.151}
SPL {X  -159.990, Y  +610.545, Z    +0.000, E1   -41.917, E3 +370988.121}
SPL {X  -159.990, Y  +615.720, Z    +0.000, E1   -41.899, E3 +371000.381}
SPL {X  -159.990, Y  +621.417, Z    +0.000, E1   -41.931, E3 +371013.818}
SPL {X  -159.990, Y  +627.900, Z    +0.000, E1   -41.914, E3 +371029.157}
SPL {X  -159.990, Y  +634.411, Z    +0.000, E1   -41.931, E3 +371044.526}
SPL {X  -159.990, Y  +641.479, Z    +0.000, E1   -41.931, E3 +371061.243}
SPL {X  -159.990, Y  +647.782, Z    +0.000, E1   -41.914, E3 +371076.165}
SPL {X  -159.990, Y  +653.094, Z    +0.000, E1   -41.905, E3 +371088.743}
SPL {X  -159.990, Y  +657.893, Z    +0.000, E1   -41.899, E3 +371100.109}
SPL {X  -159.990, Y  +662.516, Z    +0.000, E1   -41.899, E3 +371111.040}
SPL {X  -159.990, Y  +668.411, Z    +0.000, E1   -41.929, E3 +371124.934}
SPL {X  -159.968, Y  +674.139, Z    +0.000, E1   -41.898, E3 +371138.538}
SPL {X  -159.817, Y  +678.937, Z    +0.000, E1   -41.879, E3 +371150.034}
SPL {X  -159.484, Y  +684.213, Z    +0.000, E1   -41.818, E3 +371162.870}
SPL {X  -159.007, Y  +689.209, Z    +0.000, E1   -41.732, E3 +371175.175}
SPL {X  -158.327, Y  +694.511, Z    +0.000, E1   -41.622, E3 +371188.426}
SPL {X  -157.480, Y  +699.729, Z    +0.000, E1   -41.453, E3 +371201.689}
SPL {X  -156.604, Y  +704.242, Z    +0.000, E1   -41.288, E3 +371213.298}
SPL {X  -155.514, Y  +709.078, Z    +0.000, E1   -41.107, E3 +371225.851}
SPL {X  -154.232, Y  +714.035, Z    +0.000, E1   -40.861, E3 +371238.910}
SPL {X  -153.147, Y  +717.790, Z    +0.000, E1   -40.640, E3 +371248.928}
SPL {X  -151.881, Y  +721.788, Z    +0.000, E1   -40.435, E3 +371259.615}
SPL {X  -148.572, Y  +730.857, Z    +0.000, E1   -36.304, E3 +371315.824}
ENDSPLINE

SPLINE
SPL {X  -156.377, Y  +705.307, Z    +0.000, E1   -21.740, E3 +371370.073}
SPL {X  -159.301, Y  +686.331, Z    +0.000, E1   -11.648, E3 +371382.717}
SPL {X  -159.936, Y  +675.651, Z    +0.000, E1    -5.377, E3 +371386.433}
SPL {X  -159.990, Y  +670.142, Z    +0.000, E1    -1.740, E3 +371387.732}
SPL {X  -159.990, Y  +666.629, Z    +0.000, E1    +0.827, E3 +371388.382}
SPL {X  -159.990, Y  +662.407, Z    +0.000, E1    +4.406, E3 +371389.232}
SPL {X  -159.990, Y  +657.382, Z    +0.000, E1    +9.217, E3 +371390.614}
SPL {X  -159.990, Y  +653.255, Z    +0.000, E1   +13.347, E3 +371391.943}
SPL {X  -159.990, Y  +646.242, Z    +0.000, E1   +19.956, E3 +371395.017}
SPL {X  -159.990, Y  +624.365, Z    +0.000, E1   +33.860, E3 +371412.918}
SPL {X  -159.990, Y  +615.596, Z    +0.000, E1   +36.980, E3 +371422.577}
SPL {X  -159.990, Y  +586.905, Z    +0.000, E1   +41.264, E3 +371469.603}
SPL {X  -159.990, Y  +581.111, Z    +0.000, E1   +41.245, E3 +371483.657}
SPL {X  -159.990, Y  +576.269, Z    +0.000, E1   +41.239, E3 +371495.385}
SPL {X  -159.990, Y  +571.714, Z    +0.000, E1   +41.240, E3 +371506.413}
SPL {X  -159.990, Y  +567.050, Z    +0.000, E1   +41.238, E3 +371517.699}
SPL {X  -159.990, Y  +561.959, Z    +0.000, E1   +41.251, E3 +371529.998}
SPL {X  -159.990, Y  +557.719, Z    +0.000, E1   +41.226, E3 +371540.300}
SPL {X  -159.990, Y  +554.148, Z    +0.000, E1   +41.237, E3 +371548.915}
SPL {X  -159.990, Y  +548.812, Z    +0.000, E1   +41.263, E3 +371561.790}
SPL {X  -159.990, Y  +543.804, Z    +0.000, E1   +41.237, E3 +371573.955}
SPL {X  -159.990, Y  +538.952, Z    +0.000, E1   +41.247, E3 +371585.702}
SPL {X  -159.990, Y  +534.225, Z    +0.000, E1   +41.236, E3 +371597.135}
SPL {X  -159.990, Y  +529.136, Z    +0.000, E1   +41.262, E3 +371609.411}
SPL {X  -159.990, Y  +522.690, Z    +0.000, E1   +41.265, E3 +371625.011}
SPL {X  -159.990, Y  +516.698, Z    +0.000, E1   +41.259, E3 +371639.485}
SPL {X  -159.990, Y  +510.896, Z    +0.000, E1   +41.267, E3 +371653.503}
SPL {X  -159.990, Y  +505.215, Z    +0.000, E1   +41.261, E3 +371667.263}
SPL {X  -159.990, Y  +500.102, Z    +0.000, E1   +41.251, E3 +371679.646}
SPL {X  -159.990, Y  +495.023, Z    +0.000, E1   +41.263, E3 +371691.895}
SPL {X  -159.990, Y  +479.011, Z    +0.000, E1   +45.740, E3 +371701.277}
SPL {X  -159.990, Y  +471.379, Z    +0.000, E1   +46.435, E3 +371712.892}
SPL {X  -159.990, Y  +465.881, Z    +0.000, E1   +45.385, E3 +371730.495}
SPL {X  -159.990, Y  +461.571, Z    +0.000, E1   +44.440, E3 +371745.021}
SPL {X  -159.990, Y  +458.229, Z    +0.000, E1   +43.579, E3 +371757.554}
SPL {X  -159.990, Y  +453.434, Z    +0.000, E1   +43.227, E3 +371770.329}
SPL {X  -159.990, Y  +448.702, Z    +0.000, E1   +43.218, E3 +371781.051}
SPL {X  -159.990, Y  +444.476, Z    +0.000, E1   +43.219, E3 +371790.589}
SPL {X  -159.990, Y  +440.246, Z    +0.000, E1   +43.217, E3 +371800.147}
SPL {X  -159.990, Y  +434.411, Z    +0.000, E1   +43.246, E3 +371813.277}
SPL {X  -159.990, Y  +429.216, Z    +0.000, E1   +43.210, E3 +371825.049}
SPL {X  -159.990, Y  +424.433, Z    +0.000, E1   +43.237, E3 +371835.797}
SPL {X  -159.990, Y  +419.466, Z    +0.000, E1   +43.217, E3 +371847.037}
SPL {X  -159.990, Y  +414.585, Z    +0.000, E1   +43.233, E3 +371858.029}
SPL {X  -159.990, Y  +409.927, Z    +0.000, E1   +43.217, E3 +371868.560}
SPL {X  -159.990, Y  +405.428, Z    +0.000, E1   +43.230, E3 +371878.719}
SPL {X  -159.990, Y  +398.518, Z    +0.000, E1   +43.261, E3 +371894.273}
SPL {X  -159.990, Y  +392.163, Z    +0.000, E1   +43.223, E3 +371908.673}
SPL {X  -159.990, Y  +387.342, Z    +0.000, E1   +43.224, E3 +371919.550}
SPL {X  -159.990, Y  +382.548, Z    +0.000, E1   +43.224, E3 +371930.373}
SPL {X  -159.922, Y  +377.835, Z    +0.000, E1   +43.211, E3 +371941.090}
SPL {X  -159.712, Y  +373.072, Z    +0.000, E1   +43.177, E3 +371952.056}
SPL {X  -159.289, Y  +367.537, Z    +0.000, E1   +43.118, E3 +371964.968}
SPL {X  -158.730, Y  +362.464, Z    +0.000, E1   +43.003, E3 +371977.000}
SPL {X  -158.182, Y  +358.518, Z    +0.000, E1   +42.902, E3 +371986.478}
SPL {X  -157.507, Y  +354.423, Z    +0.000, E1   +42.786, E3 +371996.423}
SPL {X  -156.676, Y  +350.104, Z    +0.000, E1   +42.637, E3 +372007.029}
SPL {X  -155.807, Y  +346.154, Z    +0.000, E1   +42.470, E3 +372016.856}
SPL {X  -154.777, Y  +341.993, Z    +0.000, E1   +42.302, E3 +372027.281}
SPL {X  -153.585, Y  +337.686, Z    +0.000, E1   +42.062, E3 +372038.256}
SPL {X  -152.412, Y  +333.846, Z    +0.000, E1   +41.856, E3 +372048.099}
SPL {X  -151.009, Y  +329.651, Z    +0.000, E1   +41.581, E3 +372058.999}
SPL {X  -148.356, Y  +322.607, Z    +0.000, E1   +36.121, E3 +372119.474}
ENDSPLINE

SPLINE
SPL {X  -156.487, Y  +349.204, Z    +0.000, E1   +21.338, E3 +372174.600}
SPL {X  -159.136, Y  +365.992, Z    +0.000, E1   +12.463, E3 +372185.359}
SPL {X  -159.799, Y  +374.694, Z    +0.000, E1    +7.504, E3 +372188.462}
SPL {X  -159.976, Y  +380.404, Z    +0.000, E1    +3.959, E3 +372189.995}
SPL {X  -159.990, Y  +384.773, Z    +0.000, E1    +1.003, E3 +372190.890}
SPL {X  -159.990, Y  +387.968, Z    +0.000, E1    -1.448, E3 +372191.458}
SPL {X  -159.990, Y  +391.397, Z    +0.000, E1    -4.422, E3 +372192.082}
SPL {X  -159.990, Y  +395.864, Z    +0.000, E1    -8.712, E3 +372193.171}
SPL {X  -159.990, Y  +401.273, Z    +0.000, E1   -14.176, E3 +372194.898}
SPL {X  -159.990, Y  +411.788, Z    +0.000, E1   -23.693, E3 +372200.441}
SPL {X  -159.990, Y  +438.158, Z    +0.000, E1   -37.630, E3 +372223.718}
SPL {X  -159.990, Y  +465.724, Z    +0.000, E1   -41.883, E3 +372266.413}
SPL {X  -159.990, Y  +470.837, Z    +0.000, E1   -41.927, E3 +372278.427}
SPL {X  -159.990, Y  +477.498, Z    +0.000, E1   -41.916, E3 +372294.203}
SPL {X  -159.990, Y  +483.140, Z    +0.000, E1   -41.902, E3 +372307.559}
SPL {X  -159.990, Y  +488.618, Z    +0.000, E1   -41.913, E3 +372320.491}
SPL {X  -159.990, Y  +494.299, Z    +0.000, E1   -41.910, E3 +372333.925}
SPL {X  -159.990, Y  +499.538, Z    +0.000, E1   -41.904, E3 +372346.319}
SPL {X  -159.990, Y  +504.097, Z    +0.000, E1   -41.897, E3 +372357.108}
SPL {X  -159.990, Y  +509.413, Z    +0.000, E1   -41.921, E3 +372369.643}
SPL {X  -159.990, Y  +516.193, Z    +0.000, E1   -41.932, E3 +372385.659}
SPL {X  -159.990, Y  +521.318, Z    +0.000, E1   -41.891, E3 +372397.833}
SPL {X  -159.990, Y  +526.974, Z    +0.000, E1   -41.950, E3 +372411.122}
SPL {X  -159.990, Y  +533.758, Z    +0.000, E1   -41.910, E3 +372427.225}
SPL {X  -159.990, Y  +539.474, Z    +0.000, E1   -41.912, E3 +372440.752}
SPL {X  -159.990, Y  +546.447, Z    +0.000, E1   -41.939, E3 +372457.215}
SPL {X  -159.990, Y  +552.220, Z    +0.000, E1   -41.887, E3 +372470.949}
SPL {X  -159.990, Y  +556.952, Z    +0.000, E1   -41.911, E3 +372482.084}
SPL {X  -159.990, Y  +562.629, Z    +0.000, E1   -41.910, E3 +372495.502}
SPL {X  -159.990, Y  +567.682, Z    +0.000, E1   -41.901, E3 +372507.461}
SPL {X  -159.990, Y  +574.350, Z    +0.000, E1   -41.955, E3 +372523.147}
SPL {X  -159.990, Y  +580.118, Z    +0.000, E1   -41.891, E3 +372536.883}
SPL {X  -159.990, Y  +584.320, Z    +0.000, E1   -41.901, E3 +372546.819}
SPL {X  -159.990, Y  +589.217, Z    +0.000, E1   -41.901, E3 +372558.392}
SPL {X  -159.990, Y  +594.252, Z    +0.000, E1   -41.903, E3 +372570.307}
SPL {X  -159.990, Y  +598.793, Z    +0.000, E1   -41.896, E3 +372581.060}
SPL {X  -159.990, Y  +604.215, Z    +0.000, E1   -41.919, E3 +372593.841}
SPL {X  -159.990, Y  +610.545, Z    +0.000, E1   -41.917, E3 +372608.810}
SPL {X  -159.990, Y  +615.720, Z    +0.000, E1   -41.899, E3 +372621.071}
SPL {X  -159.990, Y  +620.005, Z    +0.000, E1   -41.900, E3 +372631.203}
SPL {X  -159.990, Y  +624.919, Z    +0.000, E1   -41.912, E3 +372642.811}
SPL {X  -159.990, Y  +630.816, Z    +0.000, E1   -41.915, E3 +372656.740}
SPL {X  -159.990, Y  +635.747, Z    +0.000, E1   -41.898, E3 +372668.418}
SPL {X  -159.990, Y  +641.479, Z    +0.000, E1   -41.931, E3 +372681.933}
SPL {X  -159.990, Y  +647.782, Z    +0.000, E1   -41.914, E3 +372696.855}
SPL {X  -159.990, Y  +653.094, Z    +0.000, E1   -41.905, E3 +372709.433}
SPL {X  -159.990, Y  +657.893, Z    +0.000, E1   -41.899, E3 +372720.798}
SPL {X  -159.990, Y  +662.516, Z    +0.000, E1   -41.899, E3 +372731.730}
SPL {X  -159.990, Y  +668.411, Z    +0.000, E1   -41.929, E3 +372745.623}
SPL {X  -159.968, Y  +674.139, Z    +0.000, E1   -41.898, E3 +372759.227}
SPL {X  -159.817, Y  +678.937, Z    +0.000, E1   -41.879, E3 +372770.724}
SPL {X  -159.484, Y  +684.213, Z    +0.000, E1   -41.818, E3 +372783.560}
SPL {X  -159.007, Y  +689.209, Z    +0.000, E1   -41.732, E3 +372795.865}
SPL {X  -158.327, Y  +694.511, Z    +0.000, E1   -41.622, E3 +372809.115}
SPL {X  -157.480, Y  +699.729, Z    +0.000, E1   -41.453, E3 +372822.378}
SPL {X  -156.604, Y  +704.242, Z    +0.000, E1   -41.288, E3 +372833.987}
SPL {X  -155.514, Y  +709.078, Z    +0.000, E1   -41.107, E3 +372846.541}
SPL {X  -154.232, Y  +714.035, Z    +0.000, E1   -40.861, E3 +372859.600}
SPL {X  -153.147, Y  +717.790, Z    +0.000, E1   -40.640, E3 +372869.618}
SPL {X  -151.881, Y  +721.788, Z    +0.000, E1   -40.435, E3 +372880.305}
SPL {X  -148.572, Y  +730.857, Z    +0.000, E1   -36.304, E3 +372936.514}
ENDSPLINE

SPLINE
SPL {X  -156.377, Y  +705.307, Z    +0.000, E1   -21.740, E3 +372990.762}
SPL {X  -159.301, Y  +686.331, Z    +0.000, E1   -11.648, E3 +373003.407}
SPL {X  -159.936, Y  +675.651, Z    +0.000, E1    -5.377, E3 +373007.123}
SPL {X  -159.990, Y  +670.142, Z    +0.000, E1    -1.740, E3 +373008.422}
SPL {X  -159.990, Y  +666.629, Z    +0.000, E1    +0.827, E3 +373009.071}
SPL {X  -159.990, Y  +662.407, Z    +0.000, E1    +4.406, E3 +373009.922}
SPL {X  -159.990, Y  +655.884, Z    +0.000, E1   +10.601, E3 +373011.787}
SPL {X  -159.990, Y  +643.833, Z    +0.000, E1   +21.883, E3 +373017.416}
SPL {X  -159.990, Y  +617.235, Z    +0.000, E1   +36.481, E3 +373041.316}
SPL {X  -159.990, Y  +586.905, Z    +0.000, E1   +41.264, E3 +373090.293}
SPL {X  -159.990, Y  +581.111, Z    +0.000, E1   +41.245, E3 +373104.347}
SPL {X  -159.990, Y  +576.269, Z    +0.000, E1   +41.239, E3 +373116.074}
SPL {X  -159.990, Y  +571.714, Z    +0.000, E1   +41.240, E3 +373127.102}
SPL {X  -159.990, Y  +567.050, Z    +0.000, E1   +41.238, E3 +373138.389}
SPL {X  -159.990, Y  +561.959, Z    +0.000, E1   +41.251, E3 +373150.688}
SPL {X  -159.990, Y  +555.553, Z    +0.000, E1   +41.273, E3 +373166.156}
SPL {X  -159.990, Y  +549.897, Z    +0.000, E1   +41.240, E3 +373179.886}
SPL {X  -159.990, Y  +544.775, Z    +0.000, E1   +41.260, E3 +373192.261}
SPL {X  -159.990, Y  +540.176, Z    +0.000, E1   +41.224, E3 +373203.469}
SPL {X  -159.990, Y  +534.009, Z    +0.000, E1   +41.300, E3 +373218.255}
SPL {X  -159.990, Y  +526.579, Z    +0.000, E1   +41.262, E3 +373236.292}
SPL {X  -159.990, Y  +521.454, Z    +0.000, E1   +41.236, E3 +373248.736}
SPL {X  -159.990, Y  +515.605, Z    +0.000, E1   +41.288, E3 +373262.776}
SPL {X  -159.990, Y  +509.898, Z    +0.000, E1   +41.246, E3 +373276.637}
SPL {X  -159.990, Y  +505.215, Z    +0.000, E1   +41.261, E3 +373287.953}
SPL {X  -159.990, Y  +500.102, Z    +0.000, E1   +41.251, E3 +373300.336}
SPL {X  -159.990, Y  +495.023, Z    +0.000, E1   +41.263, E3 +373312.585}
SPL {X  -159.990, Y  +479.011, Z    +0.000, E1   +45.740, E3 +373321.967}
SPL {X  -159.990, Y  +471.379, Z    +0.000, E1   +46.435, E3 +373333.582}
SPL {X  -159.990, Y  +465.881, Z    +0.000, E1   +45.385, E3 +373351.185}
SPL {X  -159.990, Y  +461.571, Z    +0.000, E1   +44.440, E3 +373365.710}
SPL {X  -159.990, Y  +458.229, Z    +0.000, E1   +43.579, E3 +373378.244}
SPL {X  -159.990, Y  +453.434, Z    +0.000, E1   +43.227, E3 +373391.018}
SPL {X  -159.990, Y  +448.702, Z    +0.000, E1   +43.218, E3 +373401.740}
SPL {X  -159.990, Y  +442.224, Z    +0.000, E1   +43.270, E3 +373416.290}
SPL {X  -159.990, Y  +435.724, Z    +0.000, E1   +43.218, E3 +373431.048}
SPL {X  -159.990, Y  +430.527, Z    +0.000, E1   +43.236, E3 +373442.738}
SPL {X  -159.990, Y  +424.433, Z    +0.000, E1   +43.237, E3 +373456.487}
SPL {X  -159.990, Y  +419.466, Z    +0.000, E1   +43.217, E3 +373467.726}
SPL {X  -159.990, Y  +414.585, Z    +0.000, E1   +43.233, E3 +373478.718}
SPL {X  -159.990, Y  +409.927, Z    +0.000, E1   +43.217, E3 +373489.250}
SPL {X  -159.990, Y  +405.428, Z    +0.000, E1   +43.230, E3 +373499.408}
SPL {X  -159.990, Y  +401.033, Z    +0.000, E1   +43.209, E3 +373509.363}
SPL {X  -159.990, Y  +396.968, Z    +0.000, E1   +43.221, E3 +373518.521}
SPL {X  -159.990, Y  +392.163, Z    +0.000, E1   +43.223, E3 +373529.363}
SPL {X  -159.990, Y  +387.342, Z    +0.000, E1   +43.224, E3 +373540.240}
SPL {X  -159.990, Y  +382.548, Z    +0.000, E1   +43.224, E3 +373551.063}
SPL {X  -159.922, Y  +377.835, Z    +0.000, E1   +43.211, E3 +373561.780}
SPL {X  -159.712, Y  +373.072, Z    +0.000, E1   +43.177, E3 +373572.745}
SPL {X  -159.289, Y  +367.537, Z    +0.000, E1   +43.118, E3 +373585.657}
SPL {X  -158.730, Y  +362.464, Z    +0.000, E1   +43.003, E3 +373597.689}
SPL {X  -158.182, Y  +358.518, Z    +0.000, E1   +42.902, E3 +373607.168}
SPL {X  -157.507, Y  +354.423, Z    +0.000, E1   +42.786, E3 +373617.113}
SPL {X  -156.676, Y  +350.104, Z    +0.000, E1   +42.637, E3 +373627.718}
SPL {X  -155.807, Y  +346.154, Z    +0.000, E1   +42.470, E3 +373637.545}
SPL {X  -154.777, Y  +341.993, Z    +0.000, E1   +42.302, E3 +373647.971}
SPL {X  -153.585, Y  +337.686, Z    +0.000, E1   +42.062, E3 +373658.946}
SPL {X  -152.412, Y  +333.846, Z    +0.000, E1   +41.856, E3 +373668.789}
SPL {X  -151.009, Y  +329.651, Z    +0.000, E1   +41.581, E3 +373679.688}
SPL {X  -148.356, Y  +322.607, Z    +0.000, E1   +36.121, E3 +373740.164}
ENDSPLINE

SPLINE
SPL {X  -156.487, Y  +349.204, Z    +0.000, E1   +21.338, E3 +373795.290}
SPL {X  -159.136, Y  +365.992, Z    +0.000, E1   +12.463, E3 +373806.048}
SPL {X  -159.799, Y  +374.694, Z    +0.000, E1    +7.504, E3 +373809.152}
SPL {X  -159.976, Y  +380.404, Z    +0.000, E1    +3.959, E3 +373810.685}
SPL {X  -159.990, Y  +384.773, Z    +0.000, E1    +1.003, E3 +373811.580}
SPL {X  -159.990, Y  +387.968, Z    +0.000, E1    -1.448, E3 +373812.148}
SPL {X  -159.990, Y  +391.397, Z    +0.000, E1    -4.422, E3 +373812.772}
SPL {X  -159.990, Y  +395.864, Z    +0.000, E1    -8.712, E3 +373813.860}
SPL {X  -159.990, Y  +401.273, Z    +0.000, E1   -14.176, E3 +373815.588}
SPL {X  -159.990, Y  +411.788, Z    +0.000, E1   -23.693, E3 +373821.131}
SPL {X  -159.990, Y  +438.158, Z    +0.000, E1   -37.630, E3 +373844.408}
SPL {X  -159.990, Y  +468.567, Z    +0.000, E1   -41.922, E3 +373893.752}
SPL {X  -159.990, Y  +474.616, Z    +0.000, E1   -41.909, E3 +373908.081}
SPL {X  -159.990, Y  +478.952, Z    +0.000, E1   -41.885, E3 +373918.379}
SPL {X  -159.990, Y  +484.724, Z    +0.000, E1   -41.943, E3 +373931.931}
SPL {X  -159.990, Y  +492.944, Z    +0.000, E1   -41.952, E3 +373951.350}
SPL {X  -159.990, Y  +499.538, Z    +0.000, E1   -41.904, E3 +373967.009}
SPL {X  -159.990, Y  +504.097, Z    +0.000, E1   -41.897, E3 +373977.797}
SPL {X  -159.990, Y  +509.413, Z    +0.000, E1   -41.921, E3 +373990.332}
SPL {X  -159.990, Y  +516.193, Z    +0.000, E1   -41.932, E3 +374006.349}
SPL {X  -159.990, Y  +521.318, Z    +0.000, E1   -41.891, E3 +374018.523}
SPL {X  -159.990, Y  +526.974, Z    +0.000, E1   -41.950, E3 +374031.812}
SPL {X  -159.990, Y  +533.758, Z    +0.000, E1   -41.910, E3 +374047.914}
SPL {X  -159.990, Y  +539.474, Z    +0.000, E1   -41.912, E3 +374061.442}
SPL {X  -159.990, Y  +544.879, Z    +0.000, E1   -41.899, E3 +374074.253}
SPL {X  -159.990, Y  +550.802, Z    +0.000, E1   -41.920, E3 +374088.235}
SPL {X  -159.990, Y  +556.952, Z    +0.000, E1   -41.911, E3 +374102.774}
SPL {X  -159.990, Y  +562.629, Z    +0.000, E1   -41.910, E3 +374116.192}
SPL {X  -159.990, Y  +567.682, Z    +0.000, E1   -41.901, E3 +374128.151}
SPL {X  -159.990, Y  +572.912, Z    +0.000, E1   -41.914, E3 +374140.498}
SPL {X  -159.990, Y  +578.863, Z    +0.000, E1   -41.918, E3 +374154.562}
SPL {X  -159.990, Y  +584.320, Z    +0.000, E1   -41.901, E3 +374167.509}
SPL {X  -159.990, Y  +589.217, Z    +0.000, E1   -41.901, E3 +374179.082}
SPL {X  -159.990, Y  +594.252, Z    +0.000, E1   -41.903, E3 +374190.996}
SPL {X  -159.990, Y  +600.237, Z    +0.000, E1   -41.928, E3 +374205.114}
SPL {X  -159.990, Y  +605.518, Z    +0.000, E1   -41.890, E3 +374217.652}
SPL {X  -159.990, Y  +610.545, Z    +0.000, E1   -41.917, E3 +374229.500}
SPL {X  -159.990, Y  +615.720, Z    +0.000, E1   -41.899, E3 +374241.760}
SPL {X  -159.990, Y  +621.417, Z    +0.000, E1   -41.931, E3 +374255.197}
SPL {X  -159.990, Y  +627.900, Z    +0.000, E1   -41.914, E3 +374270.537}
SPL {X  -159.990, Y  +632.270, Z    +0.000, E1   -41.887, E3 +374280.913}
SPL {X  -159.990, Y  +637.009, Z    +0.000, E1   -41.925, E3 +374292.055}
SPL {X  -159.990, Y  +642.624, Z    +0.000, E1   -41.901, E3 +374305.376}
SPL {X  -159.990, Y  +647.782, Z    +0.000, E1   -41.914, E3 +374317.544}
SPL {X  -159.990, Y  +653.094, Z    +0.000, E1   -41.905, E3 +374330.122}
SPL {X  -159.990, Y  +657.893, Z    +0.000, E1   -41.899, E3 +374341.488}
SPL {X  -159.990, Y  +662.516, Z    +0.000, E1   -41.899, E3 +374352.419}
SPL {X  -159.990, Y  +666.974, Z    +0.000, E1   -41.897, E3 +374362.964}
SPL {X  -159.984, Y  +672.859, Z    +0.000, E1   -41.934, E3 +374376.825}
SPL {X  -159.817, Y  +678.937, Z    +0.000, E1   -41.879, E3 +374391.413}
SPL {X  -159.484, Y  +684.213, Z    +0.000, E1   -41.818, E3 +374404.249}
SPL {X  -159.007, Y  +689.209, Z    +0.000, E1   -41.732, E3 +374416.554}
SPL {X  -158.327, Y  +694.511, Z    +0.000, E1   -41.622, E3 +374429.805}
SPL {X  -157.480, Y  +699.729, Z    +0.000, E1   -41.453, E3 +374443.068}
SPL {X  -156.604, Y  +704.242, Z    +0.000, E1   -41.288, E3 +374454.677}
SPL {X  -155.514, Y  +709.078, Z    +0.000, E1   -41.107, E3 +374467.230}
SPL {X  -154.232, Y  +714.035, Z    +0.000, E1   -40.861, E3 +374480.289}
SPL {X  -153.147, Y  +717.790, Z    +0.000, E1   -40.640, E3 +374490.308}
SPL {X  -151.881, Y  +721.788, Z    +0.000, E1   -40.435, E3 +374500.994}
SPL {X  -148.572, Y  +730.857, Z    +0.000, E1   -36.304, E3 +374557.203}
ENDSPLINE

SPLINE
SPL {X  -156.377, Y  +705.307, Z    +0.000, E1   -21.740, E3 +374611.452}
SPL {X  -158.965, Y  +689.585, Z    +0.000, E1   -13.405, E3 +374622.609}
SPL {X  -159.884, Y  +677.314, Z    +0.000, E1    -6.475, E3 +374627.322}
SPL {X  -159.990, Y  +670.142, Z    +0.000, E1    -1.740, E3 +374629.111}
SPL {X  -159.990, Y  +666.629, Z    +0.000, E1    +0.827, E3 +374629.761}
SPL {X  -159.990, Y  +662.407, Z    +0.000, E1    +4.406, E3 +374630.611}
SPL {X  -159.990, Y  +655.884, Z    +0.000, E1   +10.601, E3 +374632.477}
SPL {X  -159.990, Y  +643.833, Z    +0.000, E1   +21.883, E3 +374638.106}
SPL {X  -159.990, Y  +617.235, Z    +0.000, E1   +36.481, E3 +374662.006}
SPL {X  -159.990, Y  +586.905, Z    +0.000, E1   +41.264, E3 +374710.982}
SPL {X  -159.990, Y  +581.111, Z    +0.000, E1   +41.245, E3 +374725.036}
SPL {X  -159.990, Y  +576.269, Z    +0.000, E1   +41.239, E3 +374736.764}
SPL {X  -159.990, Y  +571.714, Z    +0.000, E1   +41.240, E3 +374747.792}
SPL {X  -159.990, Y  +567.050, Z    +0.000, E1   +41.238, E3 +374759.079}
SPL {X  -159.990, Y  +561.959, Z    +0.000, E1   +41.251, E3 +374771.377}
SPL {X  -159.990, Y  +557.719, Z    +0.000, E1   +41.226, E3 +374781.680}
SPL {X  -159.990, Y  +554.148, Z    +0.000, E1   +41.237, E3 +374790.295}
SPL {X  -159.990, Y  +548.812, Z    +0.000, E1   +41.263, E3 +374803.169}
SPL {X  -159.990, Y  +543.804, Z    +0.000, E1   +41.237, E3 +374815.334}
SPL {X  -159.990, Y  +538.952, Z    +0.000, E1   +41.247, E3 +374827.081}
SPL {X  -159.990, Y  +534.225, Z    +0.000, E1   +41.236, E3 +374838.515}
SPL {X  -159.990, Y  +529.136, Z    +0.000, E1   +41.262, E3 +374850.790}
SPL {X  -159.990, Y  +522.690, Z    +0.000, E1   +41.265, E3 +374866.390}
SPL {X  -159.990, Y  +516.698, Z    +0.000, E1   +41.259, E3 +374880.864}
SPL {X  -159.990, Y  +510.896, Z    +0.000, E1   +41.267, E3 +374894.882}
SPL {X  -159.990, Y  +505.215, Z    +0.000, E1   +41.261, E3 +374908.642}
SPL {X  -159.990, Y  +500.102, Z    +0.000, E1   +41.251, E3 +374921.025}
SPL {X  -159.990, Y  +495.023, Z    +0.000, E1   +41.263, E3 +374933.274}
SPL {X  -159.990, Y  +479.011, Z    +0.000, E1   +45.740, E3 +374942.656}
SPL {X  -159.990, Y  +471.379, Z    +0.000, E1   +46.435, E3 +374954.272}
SPL {X  -159.990, Y  +466.895, Z    +0.000, E1   +45.533, E3 +374968.677}
SPL {X  -159.990, Y  +462.409, Z    +0.000, E1   +44.664, E3 +374983.451}
SPL {X  -159.990, Y  +458.229, Z    +0.000, E1   +43.579, E3 +374998.934}
SPL {X  -159.990, Y  +453.434, Z    +0.000, E1   +43.227, E3 +375011.708}
SPL {X  -159.990, Y  +448.702, Z    +0.000, E1   +43.218, E3 +375022.430}
SPL {X  -159.990, Y  +444.476, Z    +0.000, E1   +43.219, E3 +375031.968}
SPL {X  -159.990, Y  +440.246, Z    +0.000, E1   +43.217, E3 +375041.526}
SPL {X  -159.990, Y  +434.411, Z    +0.000, E1   +43.246, E3 +375054.656}
SPL {X  -159.990, Y  +429.216, Z    +0.000, E1   +43.210, E3 +375066.429}
SPL {X  -159.990, Y  +424.433, Z    +0.000, E1   +43.237, E3 +375077.176}
SPL {X  -159.990, Y  +419.466, Z    +0.000, E1   +43.217, E3 +375088.416}
SPL {X  -159.990, Y  +414.585, Z    +0.000, E1   +43.233, E3 +375099.408}
SPL {X  -159.990, Y  +409.927, Z    +0.000, E1   +43.217, E3 +375109.940}
SPL {X  -159.990, Y  +405.428, Z    +0.000, E1   +43.230, E3 +375120.098}
SPL {X  -159.990, Y  +398.518, Z    +0.000, E1   +43.261, E3 +375135.652}
SPL {X  -159.990, Y  +392.163, Z    +0.000, E1   +43.223, E3 +375150.052}
SPL {X  -159.990, Y  +387.342, Z    +0.000, E1   +43.224, E3 +375160.930}
SPL {X  -159.990, Y  +382.548, Z    +0.000, E1   +43.224, E3 +375171.752}
SPL {X  -159.922, Y  +377.835, Z    +0.000, E1   +43.211, E3 +375182.469}
SPL {X  -159.712, Y  +373.072, Z    +0.000, E1   +43.177, E3 +375193.435}
SPL {X  -159.289, Y  +367.537, Z    +0.000, E1   +43.118, E3 +375206.347}
SPL {X  -158.730, Y  +362.464, Z    +0.000, E1   +43.003, E3 +375218.379}
SPL {X  -158.182, Y  +358.518, Z    +0.000, E1   +42.902, E3 +375227.857}
SPL {X  -157.507, Y  +354.423, Z    +0.000, E1   +42.786, E3 +375237.803}
SPL {X  -156.676, Y  +350.104, Z    +0.000, E1   +42.637, E3 +375248.408}
SPL {X  -155.807, Y  +346.154, Z    +0.000, E1   +42.470, E3 +375258.235}
SPL {X  -154.777, Y  +341.993, Z    +0.000, E1   +42.302, E3 +375268.660}
SPL {X  -153.585, Y  +337.686, Z    +0.000, E1   +42.062, E3 +375279.636}
SPL {X  -152.412, Y  +333.846, Z    +0.000, E1   +41.856, E3 +375289.478}
SPL {X  -151.009, Y  +329.651, Z    +0.000, E1   +41.581, E3 +375300.378}
SPL {X  -148.356, Y  +322.607, Z    +0.000, E1   +36.121, E3 +375360.854}
ENDSPLINE

SPLINE
SPL {X  -156.487, Y  +349.204, Z    +0.000, E1   +21.338, E3 +375415.979}
SPL {X  -159.136, Y  +365.992, Z    +0.000, E1   +12.463, E3 +375426.738}
SPL {X  -159.799, Y  +374.694, Z    +0.000, E1    +7.504, E3 +375429.842}
SPL {X  -159.976, Y  +380.404, Z    +0.000, E1    +3.959, E3 +375431.375}
SPL {X  -159.990, Y  +384.773, Z    +0.000, E1    +1.003, E3 +375432.269}
SPL {X  -159.990, Y  +387.968, Z    +0.000, E1    -1.448, E3 +375432.837}
SPL {X  -159.990, Y  +391.397, Z    +0.000, E1    -4.422, E3 +375433.461}
SPL {X  -159.990, Y  +395.864, Z    +0.000, E1    -8.712, E3 +375434.550}
SPL {X  -159.990, Y  +401.273, Z    +0.000, E1   -14.176, E3 +375436.277}
SPL {X  -159.990, Y  +411.788, Z    +0.000, E1   -23.693, E3 +375441.820}
SPL {X  -159.990, Y  +438.158, Z    +0.000, E1   -37.630, E3 +375465.098}
SPL {X  -159.990, Y  +468.567, Z    +0.000, E1   -41.922, E3 +375514.441}
SPL {X  -159.990, Y  +474.616, Z    +0.000, E1   -41.909, E3 +375528.771}
SPL {X  -159.990, Y  +481.610, Z    +0.000, E1   -41.947, E3 +375545.257}
SPL {X  -159.990, Y  +488.618, Z    +0.000, E1   -41.913, E3 +375561.870}
SPL {X  -159.990, Y  +494.299, Z    +0.000, E1   -41.910, E3 +375575.304}
SPL {X  -159.990, Y  +499.538, Z    +0.000, E1   -41.904, E3 +375587.698}
SPL {X  -159.990, Y  +505.259, Z    +0.000, E1   -41.922, E3 +375601.198}
SPL {X  -159.990, Y  +511.862, Z    +0.000, E1   -41.927, E3 +375616.808}
SPL {X  -159.990, Y  +517.450, Z    +0.000, E1   -41.901, E3 +375630.055}
SPL {X  -159.990, Y  +523.027, Z    +0.000, E1   -41.926, E3 +375643.200}
SPL {X  -159.990, Y  +528.611, Z    +0.000, E1   -41.900, E3 +375656.455}
SPL {X  -159.990, Y  +533.758, Z    +0.000, E1   -41.910, E3 +375668.604}
SPL {X  -159.990, Y  +539.474, Z    +0.000, E1   -41.912, E3 +375682.131}
SPL {X  -159.990, Y  +544.879, Z    +0.000, E1   -41.899, E3 +375694.943}
SPL {X  -159.990, Y  +550.802, Z    +0.000, E1   -41.920, E3 +375708.924}
SPL {X  -159.990, Y  +556.952, Z    +0.000, E1   -41.911, E3 +375723.463}
SPL {X  -159.990, Y  +562.629, Z    +0.000, E1   -41.910, E3 +375736.881}
SPL {X  -159.990, Y  +567.682, Z    +0.000, E1   -41.901, E3 +375748.840}
SPL {X  -159.990, Y  +572.912, Z    +0.000, E1   -41.914, E3 +375761.188}
SPL {X  -159.990, Y  +578.863, Z    +0.000, E1   -41.918, E3 +375775.252}
SPL {X  -159.990, Y  +584.320, Z    +0.000, E1   -41.901, E3 +375788.198}
SPL {X  -159.990, Y  +589.217, Z    +0.000, E1   -41.901, E3 +375799.771}
SPL {X  -159.990, Y  +594.252, Z    +0.000, E1   -41.903, E3 +375811.686}
SPL {X  -159.990, Y  +598.793, Z    +0.000, E1   -41.896, E3 +375822.440}
SPL {X  -159.990, Y  +604.215, Z    +0.000, E1   -41.919, E3 +375835.220}
SPL {X  -159.990, Y  +609.216, Z    +0.000, E1   -41.890, E3 +375847.088}
SPL {X  -159.990, Y  +614.570, Z    +0.000, E1   -41.926, E3 +375859.693}
SPL {X  -159.990, Y  +620.005, Z    +0.000, E1   -41.900, E3 +375872.583}
SPL {X  -159.990, Y  +624.919, Z    +0.000, E1   -41.912, E3 +375884.190}
SPL {X  -159.990, Y  +630.816, Z    +0.000, E1   -41.915, E3 +375898.119}
SPL {X  -159.990, Y  +637.009, Z    +0.000, E1   -41.925, E3 +375912.745}
SPL {X  -159.990, Y  +642.624, Z    +0.000, E1   -41.901, E3 +375926.065}
SPL {X  -159.990, Y  +647.782, Z    +0.000, E1   -41.914, E3 +375938.234}
SPL {X  -159.990, Y  +653.094, Z    +0.000, E1   -41.905, E3 +375950.812}
SPL {X  -159.990, Y  +657.893, Z    +0.000, E1   -41.899, E3 +375962.178}
SPL {X  -159.990, Y  +662.516, Z    +0.000, E1   -41.899, E3 +375973.109}
SPL {X  -159.990, Y  +666.974, Z    +0.000, E1   -41.897, E3 +375983.653}
SPL {X  -159.984, Y  +672.859, Z    +0.000, E1   -41.934, E3 +375997.515}
SPL {X  -159.817, Y  +678.937, Z    +0.000, E1   -41.879, E3 +376012.103}
SPL {X  -159.484, Y  +684.213, Z    +0.000, E1   -41.818, E3 +376024.939}
SPL {X  -159.007, Y  +689.209, Z    +0.000, E1   -41.732, E3 +376037.244}
SPL {X  -158.327, Y  +694.511, Z    +0.000, E1   -41.622, E3 +376050.495}
SPL {X  -157.480, Y  +699.729, Z    +0.000, E1   -41.453, E3 +376063.758}
SPL {X  -156.604, Y  +704.242, Z    +0.000, E1   -41.288, E3 +376075.367}
SPL {X  -155.514, Y  +709.078, Z    +0.000, E1   -41.107, E3 +376087.920}
SPL {X  -154.232, Y  +714.035, Z    +0.000, E1   -40.861, E3 +376100.979}
SPL {X  -153.147, Y  +717.790, Z    +0.000, E1   -40.640, E3 +376110.997}
SPL {X  -151.881, Y  +721.788, Z    +0.000, E1   -40.435, E3 +376121.684}
SPL {X  -148.572, Y  +730.857, Z    +0.000, E1   -36.304, E3 +376177.893}
ENDSPLINE

SPLINE
SPL {X  -156.377, Y  +705.307, Z    +0.000, E1   -21.740, E3 +376232.142}
SPL {X  -158.965, Y  +689.585, Z    +0.000, E1   -13.405, E3 +376243.299}
SPL {X  -159.884, Y  +677.314, Z    +0.000, E1    -6.475, E3 +376248.012}
SPL {X  -159.990, Y  +670.142, Z    +0.000, E1    -1.740, E3 +376249.801}
SPL {X  -159.990, Y  +666.629, Z    +0.000, E1    +0.827, E3 +376250.451}
SPL {X  -159.990, Y  +662.407, Z    +0.000, E1    +4.406, E3 +376251.301}
SPL {X  -159.990, Y  +655.884, Z    +0.000, E1   +10.601, E3 +376253.166}
SPL {X  -159.990, Y  +643.833, Z    +0.000, E1   +21.883, E3 +376258.796}
SPL {X  -159.990, Y  +617.235, Z    +0.000, E1   +36.481, E3 +376282.696}
SPL {X  -159.990, Y  +586.905, Z    +0.000, E1   +41.264, E3 +376331.672}
SPL {X  -159.990, Y  +581.111, Z    +0.000, E1   +41.245, E3 +376345.726}
SPL {X  -159.990, Y  +576.269, Z    +0.000, E1   +41.239, E3 +376357.454}
SPL {X  -159.990, Y  +571.714, Z    +0.000, E1   +41.240, E3 +376368.482}
SPL {X  -159.990, Y  +567.050, Z    +0.000, E1   +41.238, E3 +376379.768}
SPL {X  -159.990, Y  +561.959, Z    +0.000, E1   +41.251, E3 +376392.067}
SPL {X  -159.990, Y  +557.719, Z    +0.000, E1   +41.226, E3 +376402.369}
SPL {X  -159.990, Y  +554.148, Z    +0.000, E1   +41.237, E3 +376410.984}
SPL {X  -159.990, Y  +548.812, Z    +0.000, E1   +41.263, E3 +376423.859}
SPL {X  -159.990, Y  +543.804, Z    +0.000, E1   +41.237, E3 +376436.024}
SPL {X  -159.990, Y  +538.952, Z    +0.000, E1   +41.247, E3 +376447.771}
SPL {X  -159.990, Y  +534.225, Z    +0.000, E1   +41.236, E3 +376459.204}
SPL {X  -159.990, Y  +529.136, Z    +0.000, E1   +41.262, E3 +376471.480}
SPL {X  -159.990, Y  +522.690, Z    +0.000, E1   +41.265, E3 +376487.080}
SPL {X  -159.990, Y  +516.698, Z    +0.000, E1   +41.259, E3 +376501.554}
SPL {X  -159.990, Y  +510.896, Z    +0.000, E1   +41.267, E3 +376515.572}
SPL {X  -159.990, Y  +505.215, Z    +0.000, E1   +41.261, E3 +376529.332}
SPL {X  -159.990, Y  +500.102, Z    +0.000, E1   +41.251, E3 +376541.715}
SPL {X  -159.990, Y  +495.023, Z    +0.000, E1   +41.263, E3 +376553.964}
SPL {X  -159.990, Y  +479.011, Z    +0.000, E1   +45.740, E3 +376563.346}
SPL {X  -159.990, Y  +471.379, Z    +0.000, E1   +46.435, E3 +376574.961}
SPL {X  -159.990, Y  +466.895, Z    +0.000, E1   +45.533, E3 +376589.366}
SPL {X  -159.990, Y  +462.409, Z    +0.000, E1   +44.664, E3 +376604.141}
SPL {X  -159.990, Y  +458.229, Z    +0.000, E1   +43.579, E3 +376619.623}
SPL {X  -159.990, Y  +453.434, Z    +0.000, E1   +43.227, E3 +376632.398}
SPL {X  -159.990, Y  +448.702, Z    +0.000, E1   +43.218, E3 +376643.120}
SPL {X  -159.990, Y  +444.476, Z    +0.000, E1   +43.219, E3 +376652.658}
SPL {X  -159.990, Y  +440.246, Z    +0.000, E1   +43.217, E3 +376662.215}
SPL {X  -159.990, Y  +434.411, Z    +0.000, E1   +43.246, E3 +376675.346}
SPL {X  -159.990, Y  +429.216, Z    +0.000, E1   +43.210, E3 +376687.118}
SPL {X  -159.990, Y  +424.433, Z    +0.000, E1   +43.237, E3 +376697.866}
SPL {X  -159.990, Y  +419.466, Z    +0.000, E1   +43.217, E3 +376709.106}
SPL {X  -159.990, Y  +414.585, Z    +0.000, E1   +43.233, E3 +376720.098}
SPL {X  -159.990, Y  +409.927, Z    +0.000, E1   +43.217, E3 +376730.629}
SPL {X  -159.990, Y  +405.428, Z    +0.000, E1   +43.230, E3 +376740.788}
SPL {X  -159.990, Y  +398.518, Z    +0.000, E1   +43.261, E3 +376756.342}
SPL {X  -159.990, Y  +392.163, Z    +0.000, E1   +43.223, E3 +376770.742}
SPL {X  -159.990, Y  +387.342, Z    +0.000, E1   +43.224, E3 +376781.619}
SPL {X  -159.990, Y  +382.548, Z    +0.000, E1   +43.224, E3 +376792.442}
SPL {X  -159.922, Y  +377.835, Z    +0.000, E1   +43.211, E3 +376803.159}
SPL {X  -159.712, Y  +373.072, Z    +0.000, E1   +43.177, E3 +376814.125}
SPL {X  -159.289, Y  +367.537, Z    +0.000, E1   +43.118, E3 +376827.037}
SPL {X  -158.730, Y  +362.464, Z    +0.000, E1   +43.003, E3 +376839.069}
SPL {X  -158.182, Y  +358.518, Z    +0.000, E1   +42.902, E3 +376848.547}
SPL {X  -157.507, Y  +354.423, Z    +0.000, E1   +42.786, E3 +376858.492}
SPL {X  -156.676, Y  +350.104, Z    +0.000, E1   +42.637, E3 +376869.098}
SPL {X  -155.807, Y  +346.154, Z    +0.000, E1   +42.470, E3 +376878.925}
SPL {X  -154.777, Y  +341.993, Z    +0.000, E1   +42.302, E3 +376889.350}
SPL {X  -153.585, Y  +337.686, Z    +0.000, E1   +42.062, E3 +376900.325}
SPL {X  -152.412, Y  +333.846, Z    +0.000, E1   +41.856, E3 +376910.168}
SPL {X  -151.009, Y  +329.651, Z    +0.000, E1   +41.581, E3 +376921.068}
SPL {X  -148.356, Y  +322.607, Z    +0.000, E1   +36.121, E3 +376981.543}
ENDSPLINE

